LIN {X 0,Y 519.918,Z 580.66,A -85,B 0,C 180,E1 4894.132,E2 4894.132} C_VEL
LIN {X 0,Y 514.444,Z 580.66,A -85,B 0,C 180,E1 4896.247,E2 4896.247} C_VEL
LIN {X 0,Y 514.337,Z 580.66,A -85,B 0,C 180,E1 4896.492,E2 4896.492} C_VEL
LIN {X 0,Y 514.405,Z 580.66,A -85,B 0,C 180,E1 4902.622,E2 4902.622} C_VEL
LIN {X 0,Y 514.476,Z 580.66,A -85,B 0,C 180,E1 4907.4,E2 4907.4} C_VEL
LIN {X 0,Y 514.455,Z 580.66,A -85,B 0,C 180,E1 4912.61,E2 4912.61} C_VEL
LIN {X 0,Y 514.587,Z 580.66,A -85,B 0,C 180,E1 4919.328,E2 4919.328} C_VEL
LIN {X 0,Y 526.153,Z 611.087,A -85,B 0,C 180,E1 4920.404,E2 4920.404} C_VEL
LIN {X 0,Y 525.371,Z 668.245,A -85,B 0,C 180,E1 4921.362,E2 4921.362} C_VEL
LIN {X 0,Y 524.09,Z 703.782,A -85,B 0,C 180,E1 4922.574,E2 4922.574} C_VEL
LIN {X 0,Y 522.217,Z 738.252,A -85,B 0,C 180,E1 4924.451,E2 4924.451} C_VEL
LIN {X 0,Y 520.217,Z 769.927,A -85,B 0,C 180,E1 4926.884,E2 4926.884} C_VEL
LIN {X 0,Y 518.339,Z 798.982,A -85,B 0,C 180,E1 4929.926,E2 4929.926} C_VEL
LIN {X 0,Y 516.846,Z 823.631,A -85,B 0,C 180,E1 4933.403,E2 4933.403} C_VEL
LIN {X 0,Y 515.936,Z 843.713,A -85,B 0,C 180,E1 4937.284,E2 4937.284} C_VEL
LIN {X 0,Y 515.52,Z 857.455,A -85,B 0,C 180,E1 4941.129,E2 4941.129} C_VEL
LIN {X 0,Y 515.31,Z 865.962,A -85,B 0,C 180,E1 4944.942,E2 4944.942} C_VEL
LIN {X 0,Y 515.232,Z 869.509,A -85,B 0,C 180,E1 4948.315,E2 4948.315} C_VEL
LIN {X 0,Y 515.241,Z 868.974,A -85,B 0,C 180,E1 4952.558,E2 4952.558} C_VEL
LIN {X 0,Y 515.34,Z 862.769,A -85,B 0,C 180,E1 4956.747,E2 4956.747} C_VEL
LIN {X 0,Y 515.644,Z 851.662,A -85,B 0,C 180,E1 4960.67,E2 4960.67} C_VEL
LIN {X 0,Y 516.365,Z 834.554,A -85,B 0,C 180,E1 4964.646,E2 4964.646} C_VEL
LIN {X 0,Y 517.565,Z 811.69,A -85,B 0,C 180,E1 4968.416,E2 4968.416} C_VEL
LIN {X 0,Y 519.291,Z 784.441,A -85,B 0,C 180,E1 4971.705,E2 4971.705} C_VEL
LIN {X 0,Y 521.3,Z 753.854,A -85,B 0,C 180,E1 4974.446,E2 4974.446} C_VEL
LIN {X 0,Y 523.322,Z 718.255,A -85,B 0,C 180,E1 4976.729,E2 4976.729} C_VEL
LIN {X 0,Y 524.952,Z 684.31,A -85,B 0,C 180,E1 4978.166,E2 4978.166} C_VEL
LIN {X 0,Y 525.974,Z 647.659,A -85,B 0,C 180,E1 4979.056,E2 4979.056} C_VEL
LIN {X 0,Y 525.542,Z 607.493,A -85,B 0,C 180,E1 4979.68,E2 4979.68} C_VEL
LIN {X 0,Y 514.561,Z 580.66,A -85,B 0,C 180,E1 4980.717,E2 4980.717} C_VEL
LIN {X 0,Y 514.384,Z 580.66,A -85,B 0,C 180,E1 4986.061,E2 4986.061} C_VEL
LIN {X 0,Y 514.383,Z 580.66,A -85,B 0,C 180,E1 4992.628,E2 4992.628} C_VEL
LIN {X 0,Y 514.482,Z 580.66,A -85,B 0,C 180,E1 4997.409,E2 4997.409} C_VEL
LIN {X 0,Y 514.444,Z 580.66,A -85,B 0,C 180,E1 5002.616,E2 5002.616} C_VEL
LIN {X 0,Y 514.468,Z 580.66,A -85,B 0,C 180,E1 5008.584,E2 5008.584} C_VEL
LIN {X 0,Y 514.582,Z 580.66,A -85,B 0,C 180,E1 5013.816,E2 5013.816} C_VEL
LIN {X 0,Y 514.736,Z 580.66,A -85,B 0,C 180,E1 5020.255,E2 5020.255} C_VEL
LIN {X 0,Y 514.546,Z 580.66,A -85,B 0,C 180,E1 5026.162,E2 5026.162} C_VEL
LIN {X 0,Y 514.797,Z 580.66,A -85,B 0,C 180,E1 5031.549,E2 5031.549} C_VEL
LIN {X 0,Y 514.928,Z 580.66,A -85,B 0,C 180,E1 5036.633,E2 5036.633} C_VEL
LIN {X 0,Y 514.976,Z 580.66,A -85,B 0,C 180,E1 5041.689,E2 5041.689} C_VEL
LIN {X 0,Y 514.853,Z 580.66,A -85,B 0,C 180,E1 5046.76,E2 5046.76} C_VEL
LIN {X 0,Y 514.756,Z 580.66,A -85,B 0,C 180,E1 5051.886,E2 5051.886} C_VEL
LIN {X 0,Y 514.721,Z 580.66,A -85,B 0,C 180,E1 5057.111,E2 5057.111} C_VEL
LIN {X 0,Y 514.634,Z 580.66,A -85,B 0,C 180,E1 5062.491,E2 5062.491} C_VEL
LIN {X 0,Y 514.5,Z 580.66,A -85,B 0,C 180,E1 5068.094,E2 5068.094} C_VEL
LIN {X 0,Y 514.512,Z 580.66,A -85,B 0,C 180,E1 5073.999,E2 5073.999} C_VEL
LIN {X 0,Y 514.466,Z 580.66,A -85,B 0,C 180,E1 5080.082,E2 5080.082} C_VEL
LIN {X 0,Y 514.257,Z 580.66,A -85,B 0,C 180,E1 5085.045,E2 5085.045} C_VEL
LIN {X 0,Y 514.476,Z 580.66,A -85,B 0,C 180,E1 5089.927,E2 5089.927} C_VEL
LIN {X 0,Y 514.559,Z 580.66,A -85,B 0,C 180,E1 5096.012,E2 5096.012} C_VEL
LIN {X 0,Y 514.48,Z 580.66,A -85,B 0,C 180,E1 5101.998,E2 5101.998} C_VEL
LIN {X 0,Y 514.717,Z 581.391,A -85,B 0,C 180,E1 5106.325,E2 5106.325} C_VEL
LIN {X 0,Y 522.294,Z 605.692,A -85,B 0,C 180,E1 5108.079,E2 5108.079} C_VEL
LIN {X 0,Y 520.619,Z 636.027,A -85,B 0,C 180,E1 5110.242,E2 5110.242} C_VEL
LIN {X 0,Y 518.756,Z 661.49,A -85,B 0,C 180,E1 5112.836,E2 5112.836} C_VEL
LIN {X 0,Y 517.145,Z 684.027,A -85,B 0,C 180,E1 5116.042,E2 5116.042} C_VEL
LIN {X 0,Y 516.14,Z 701.171,A -85,B 0,C 180,E1 5119.522,E2 5119.522} C_VEL
LIN {X 0,Y 515.634,Z 713.151,A -85,B 0,C 180,E1 5123.257,E2 5123.257} C_VEL
LIN {X 0,Y 515.417,Z 719.891,A -85,B 0,C 180,E1 5127.222,E2 5127.222} C_VEL
LIN {X 0,Y 515.407,Z 721.257,A -85,B 0,C 180,E1 5130.002,E2 5130.002} C_VEL
LIN {X 0,Y 515.483,Z 718.032,A -85,B 0,C 180,E1 5134.212,E2 5134.212} C_VEL
LIN {X 0,Y 515.769,Z 709.434,A -85,B 0,C 180,E1 5138.017,E2 5138.017} C_VEL
LIN {X 0,Y 516.485,Z 694.755,A -85,B 0,C 180,E1 5141.843,E2 5141.843} C_VEL
LIN {X 0,Y 517.776,Z 675.211,A -85,B 0,C 180,E1 5145.26,E2 5145.26} C_VEL
LIN {X 0,Y 519.442,Z 651.913,A -85,B 0,C 180,E1 5148.152,E2 5148.152} C_VEL
LIN {X 0,Y 521.339,Z 625.142,A -85,B 0,C 180,E1 5150.533,E2 5150.533} C_VEL
LIN {X 0,Y 521.725,Z 602.202,A -85,B 0,C 180,E1 5152.079,E2 5152.079} C_VEL
LIN {X 0,Y 514.687,Z 580.66,A -85,B 0,C 180,E1 5153.646,E2 5153.646} C_VEL
LIN {X 0,Y 514.448,Z 580.66,A -85,B 0,C 180,E1 5160.022,E2 5160.022} C_VEL
LIN {X 0,Y 514.456,Z 580.66,A -85,B 0,C 180,E1 5166.059,E2 5166.059} C_VEL
LIN {X 0,Y 514.454,Z 580.66,A -85,B 0,C 180,E1 5170.352,E2 5170.352} C_VEL
LIN {X 0,Y 514.383,Z 580.66,A -85,B 0,C 180,E1 5175.05,E2 5175.05} C_VEL
LIN {X 0,Y 514.436,Z 580.66,A -85,B 0,C 180,E1 5179.927,E2 5179.927} C_VEL
LIN {X 0,Y 514.363,Z 580.66,A -85,B 0,C 180,E1 5185.989,E2 5185.989} C_VEL
LIN {X 0,Y 514.485,Z 580.66,A -85,B 0,C 180,E1 5191.99,E2 5191.99} C_VEL
LIN {X 0,Y 514.66,Z 580.66,A -85,B 0,C 180,E1 5197.51,E2 5197.51} C_VEL
LIN {X 0,Y 514.744,Z 580.66,A -85,B 0,C 180,E1 5202.89,E2 5202.89} C_VEL
LIN {X 0,Y 514.749,Z 580.66,A -85,B 0,C 180,E1 5209.831,E2 5209.831} C_VEL
LIN {X 0,Y 514.979,Z 580.66,A -85,B 0,C 180,E1 5214.935,E2 5214.935} C_VEL
LIN {X 0,Y 515.032,Z 580.66,A -85,B 0,C 180,E1 5219.995,E2 5219.995} C_VEL
LIN {X 0,Y 514.945,Z 580.66,A -85,B 0,C 180,E1 5225.056,E2 5225.056} C_VEL
LIN {X 0,Y 514.862,Z 580.66,A -85,B 0,C 180,E1 5230.158,E2 5230.158} C_VEL
LIN {X 0,Y 514.764,Z 580.66,A -85,B 0,C 180,E1 5235.345,E2 5235.345} C_VEL
LIN {X 0,Y 514.669,Z 580.66,A -85,B 0,C 180,E1 5240.666,E2 5240.666} C_VEL
LIN {X 0,Y 514.547,Z 580.66,A -85,B 0,C 180,E1 5246.186,E2 5246.186} C_VEL
LIN {X 0,Y 514.468,Z 580.66,A -85,B 0,C 180,E1 5251.981,E2 5251.981} C_VEL
LIN {X 0,Y 514.337,Z 580.66,A -85,B 0,C 180,E1 5256.492,E2 5256.492} C_VEL
LIN {X 0,Y 513.032,Z 580.66,A -85,B 0,C 180,E1 5257.458,E2 5257.458} C_VEL
LIN {X 0,Y 506.4,Z 580.66,A -85,B 0,C 180,E1 5260.09,E2 5260.09} C_VEL
LIN {X 0,Y 506.318,Z 580.66,A -85,B 0,C 180,E1 5260.34,E2 5260.34} C_VEL
LIN {X 0,Y 506.489,Z 580.66,A -85,B 0,C 180,E1 5266.563,E2 5266.563} C_VEL
LIN {X 0,Y 506.522,Z 580.66,A -85,B 0,C 180,E1 5273.285,E2 5273.285} C_VEL
LIN {X 0,Y 506.623,Z 580.66,A -85,B 0,C 180,E1 5278.911,E2 5278.911} C_VEL
LIN {X 0,Y 518.95,Z 611.439,A -85,B 0,C 180,E1 5280.047,E2 5280.047} C_VEL
LIN {X 0,Y 518.154,Z 666.942,A -85,B 0,C 180,E1 5280.995,E2 5280.995} C_VEL
LIN {X 0,Y 516.676,Z 704.173,A -85,B 0,C 180,E1 5282.276,E2 5282.276} C_VEL
LIN {X 0,Y 514.856,Z 739.728,A -85,B 0,C 180,E1 5284.176,E2 5284.176} C_VEL
LIN {X 0,Y 512.715,Z 771.394,A -85,B 0,C 180,E1 5286.662,E2 5286.662} C_VEL
LIN {X 0,Y 510.658,Z 800.734,A -85,B 0,C 180,E1 5289.837,E2 5289.837} C_VEL
LIN {X 0,Y 509.045,Z 824.956,A -85,B 0,C 180,E1 5293.364,E2 5293.364} C_VEL
LIN {X 0,Y 508.133,Z 843.713,A -85,B 0,C 180,E1 5297.086,E2 5297.086} C_VEL
LIN {X 0,Y 507.653,Z 857.481,A -85,B 0,C 180,E1 5301,E2 5301} C_VEL
LIN {X 0,Y 507.414,Z 865.961,A -85,B 0,C 180,E1 5304.863,E2 5304.863} C_VEL
LIN {X 0,Y 507.351,Z 869.51,A -85,B 0,C 180,E1 5308.288,E2 5308.288} C_VEL
LIN {X 0,Y 507.414,Z 869.512,A -85,B 0,C 180,E1 5311.708,E2 5311.708} C_VEL
LIN {X 0,Y 507.418,Z 864.456,A -85,B 0,C 180,E1 5315.993,E2 5315.993} C_VEL
LIN {X 0,Y 507.659,Z 854.965,A -85,B 0,C 180,E1 5319.832,E2 5319.832} C_VEL
LIN {X 0,Y 508.272,Z 839.833,A -85,B 0,C 180,E1 5323.785,E2 5323.785} C_VEL
LIN {X 0,Y 509.412,Z 818.483,A -85,B 0,C 180,E1 5327.691,E2 5327.691} C_VEL
LIN {X 0,Y 511.093,Z 793.355,A -85,B 0,C 180,E1 5331.057,E2 5331.057} C_VEL
LIN {X 0,Y 513.309,Z 763.038,A -85,B 0,C 180,E1 5334.075,E2 5334.075} C_VEL
LIN {X 0,Y 515.376,Z 731.713,A -85,B 0,C 180,E1 5336.323,E2 5336.323} C_VEL
LIN {X 0,Y 517.147,Z 695.545,A -85,B 0,C 180,E1 5338.079,E2 5338.079} C_VEL
LIN {X 0,Y 518.453,Z 658.867,A -85,B 0,C 180,E1 5339.19,E2 5339.19} C_VEL
LIN {X 0,Y 518.382,Z 609.73,A -85,B 0,C 180,E1 5340.008,E2 5340.008} C_VEL
LIN {X 0,Y 506.626,Z 580.66,A -85,B 0,C 180,E1 5341.084,E2 5341.084} C_VEL
LIN {X 0,Y 506.455,Z 580.66,A -85,B 0,C 180,E1 5346.717,E2 5346.717} C_VEL
LIN {X 0,Y 506.434,Z 580.66,A -85,B 0,C 180,E1 5353.438,E2 5353.438} C_VEL
LIN {X 0,Y 506.488,Z 580.66,A -85,B 0,C 180,E1 5358.886,E2 5358.886} C_VEL
LIN {X 0,Y 506.475,Z 580.66,A -85,B 0,C 180,E1 5365.397,E2 5365.397} C_VEL
LIN {X 0,Y 506.544,Z 580.66,A -85,B 0,C 180,E1 5371.436,E2 5371.436} C_VEL
LIN {X 0,Y 506.713,Z 580.66,A -85,B 0,C 180,E1 5377.854,E2 5377.854} C_VEL
LIN {X 0,Y 506.883,Z 580.66,A -85,B 0,C 180,E1 5382.899,E2 5382.899} C_VEL
LIN {X 0,Y 506.859,Z 580.66,A -85,B 0,C 180,E1 5389.68,E2 5389.68} C_VEL
LIN {X 0,Y 507.037,Z 580.66,A -85,B 0,C 180,E1 5394.865,E2 5394.865} C_VEL
LIN {X 0,Y 507.151,Z 580.66,A -85,B 0,C 180,E1 5400.005,E2 5400.005} C_VEL
LIN {X 0,Y 507.026,Z 580.66,A -85,B 0,C 180,E1 5405.144,E2 5405.144} C_VEL
LIN {X 0,Y 506.922,Z 580.66,A -85,B 0,C 180,E1 5410.328,E2 5410.328} C_VEL
LIN {X 0,Y 506.825,Z 580.66,A -85,B 0,C 180,E1 5415.601,E2 5415.601} C_VEL
LIN {X 0,Y 506.725,Z 580.66,A -85,B 0,C 180,E1 5421.016,E2 5421.016} C_VEL
LIN {X 0,Y 506.598,Z 580.66,A -85,B 0,C 180,E1 5426.639,E2 5426.639} C_VEL
LIN {X 0,Y 506.565,Z 580.66,A -85,B 0,C 180,E1 5432.552,E2 5432.552} C_VEL
LIN {X 0,Y 506.585,Z 580.66,A -85,B 0,C 180,E1 5436.714,E2 5436.714} C_VEL
LIN {X 0,Y 506.392,Z 580.66,A -85,B 0,C 180,E1 5441.632,E2 5441.632} C_VEL
LIN {X 0,Y 506.398,Z 580.66,A -85,B 0,C 180,E1 5448.377,E2 5448.377} C_VEL
LIN {X 0,Y 506.644,Z 580.66,A -85,B 0,C 180,E1 5453.798,E2 5453.798} C_VEL
LIN {X 0,Y 506.605,Z 580.66,A -85,B 0,C 180,E1 5460.085,E2 5460.085} C_VEL
LIN {X 0,Y 506.739,Z 581.087,A -85,B 0,C 180,E1 5465.795,E2 5465.795} C_VEL
LIN {X 0,Y 515.338,Z 608.137,A -85,B 0,C 180,E1 5467.767,E2 5467.767} C_VEL
LIN {X 0,Y 513.45,Z 638.063,A -85,B 0,C 180,E1 5469.955,E2 5469.955} C_VEL
LIN {X 0,Y 511.415,Z 663.071,A -85,B 0,C 180,E1 5472.559,E2 5472.559} C_VEL
LIN {X 0,Y 509.742,Z 684.128,A -85,B 0,C 180,E1 5475.585,E2 5475.585} C_VEL
LIN {X 0,Y 508.574,Z 700.614,A -85,B 0,C 180,E1 5478.898,E2 5478.898} C_VEL
LIN {X 0,Y 507.916,Z 713.339,A -85,B 0,C 180,E1 5482.723,E2 5482.723} C_VEL
LIN {X 0,Y 507.689,Z 720.49,A -85,B 0,C 180,E1 5486.582,E2 5486.582} C_VEL
LIN {X 0,Y 507.605,Z 722.443,A -85,B 0,C 180,E1 5490.002,E2 5490.002} C_VEL
LIN {X 0,Y 507.69,Z 719.247,A -85,B 0,C 180,E1 5494.277,E2 5494.277} C_VEL
LIN {X 0,Y 508.033,Z 710.734,A -85,B 0,C 180,E1 5498.14,E2 5498.14} C_VEL
LIN {X 0,Y 508.862,Z 696.187,A -85,B 0,C 180,E1 5502.023,E2 5502.023} C_VEL
LIN {X 0,Y 510.322,Z 676.833,A -85,B 0,C 180,E1 5505.488,E2 5505.488} C_VEL
LIN {X 0,Y 512.3,Z 652.382,A -85,B 0,C 180,E1 5508.573,E2 5508.573} C_VEL
LIN {X 0,Y 514.331,Z 625.587,A -85,B 0,C 180,E1 5510.965,E2 5510.965} C_VEL
LIN {X 0,Y 514.91,Z 605.372,A -85,B 0,C 180,E1 5512.348,E2 5512.348} C_VEL
LIN {X 0,Y 506.754,Z 580.66,A -85,B 0,C 180,E1 5514.15,E2 5514.15} C_VEL
LIN {X 0,Y 506.533,Z 580.66,A -85,B 0,C 180,E1 5520.541,E2 5520.541} C_VEL
LIN {X 0,Y 506.559,Z 580.66,A -85,B 0,C 180,E1 5526.712,E2 5526.712} C_VEL
LIN {X 0,Y 506.415,Z 580.66,A -85,B 0,C 180,E1 5533.445,E2 5533.445} C_VEL
LIN {X 0,Y 506.445,Z 580.66,A -85,B 0,C 180,E1 5538.869,E2 5538.869} C_VEL
LIN {X 0,Y 506.451,Z 580.66,A -85,B 0,C 180,E1 5545.383,E2 5545.383} C_VEL
LIN {X 0,Y 506.509,Z 580.66,A -85,B 0,C 180,E1 5551.423,E2 5551.423} C_VEL
LIN {X 0,Y 506.755,Z 580.66,A -85,B 0,C 180,E1 5557.851,E2 5557.851} C_VEL
LIN {X 0,Y 506.834,Z 580.66,A -85,B 0,C 180,E1 5562.927,E2 5562.927} C_VEL
LIN {X 0,Y 506.849,Z 580.66,A -85,B 0,C 180,E1 5569.67,E2 5569.67} C_VEL
LIN {X 0,Y 507.071,Z 580.66,A -85,B 0,C 180,E1 5574.856,E2 5574.856} C_VEL
LIN {X 0,Y 507.152,Z 580.66,A -85,B 0,C 180,E1 5579.995,E2 5579.995} C_VEL
LIN {X 0,Y 507.031,Z 580.66,A -85,B 0,C 180,E1 5585.135,E2 5585.135} C_VEL
LIN {X 0,Y 506.935,Z 580.66,A -85,B 0,C 180,E1 5590.318,E2 5590.318} C_VEL
LIN {X 0,Y 506.83,Z 580.66,A -85,B 0,C 180,E1 5595.591,E2 5595.591} C_VEL
LIN {X 0,Y 506.724,Z 580.66,A -85,B 0,C 180,E1 5601.006,E2 5601.006} C_VEL
LIN {X 0,Y 506.603,Z 580.66,A -85,B 0,C 180,E1 5606.629,E2 5606.629} C_VEL
LIN {X 0,Y 506.484,Z 580.66,A -85,B 0,C 180,E1 5612.547,E2 5612.547} C_VEL
LIN {X 0,Y 506.454,Z 580.66,A -85,B 0,C 180,E1 5616.713,E2 5616.713} C_VEL
LIN {X 0,Y 506.318,Z 580.66,A -85,B 0,C 180,E1 5620.34,E2 5620.34} C_VEL
LIN {X 0,Y 503.848,Z 580.66,A -85,B 0,C 180,E1 5621.801,E2 5621.801} C_VEL
LIN {X 0,Y 498.614,Z 580.66,A -85,B 0,C 180,E1 5623.992,E2 5623.992} C_VEL
LIN {X 0,Y 498.541,Z 580.66,A -85,B 0,C 180,E1 5624.245,E2 5624.245} C_VEL
LIN {X 0,Y 498.526,Z 580.66,A -85,B 0,C 180,E1 5630.372,E2 5630.372} C_VEL
LIN {X 0,Y 498.577,Z 580.66,A -85,B 0,C 180,E1 5636.864,E2 5636.864} C_VEL
LIN {X 0,Y 498.734,Z 581.255,A -85,B 0,C 180,E1 5638.488,E2 5638.488} C_VEL
LIN {X 0,Y 511.793,Z 613.809,A -85,B 0,C 180,E1 5639.711,E2 5639.711} C_VEL
LIN {X 0,Y 510.896,Z 666.664,A -85,B 0,C 180,E1 5640.644,E2 5640.644} C_VEL
LIN {X 0,Y 509.253,Z 703.957,A -85,B 0,C 180,E1 5641.957,E2 5641.957} C_VEL
LIN {X 0,Y 507.211,Z 741.098,A -85,B 0,C 180,E1 5643.995,E2 5643.995} C_VEL
LIN {X 0,Y 505.142,Z 773.341,A -85,B 0,C 180,E1 5646.509,E2 5646.509} C_VEL
LIN {X 0,Y 503.055,Z 800.734,A -85,B 0,C 180,E1 5649.519,E2 5649.519} C_VEL
LIN {X 0,Y 501.323,Z 824.954,A -85,B 0,C 180,E1 5653.1,E2 5653.1} C_VEL
LIN {X 0,Y 500.313,Z 843.712,A -85,B 0,C 180,E1 5656.88,E2 5656.88} C_VEL
LIN {X 0,Y 499.77,Z 857.604,A -85,B 0,C 180,E1 5660.904,E2 5660.904} C_VEL
LIN {X 0,Y 499.526,Z 865.961,A -85,B 0,C 180,E1 5664.781,E2 5664.781} C_VEL
LIN {X 0,Y 499.464,Z 869.509,A -85,B 0,C 180,E1 5668.261,E2 5668.261} C_VEL
LIN {X 0,Y 499.537,Z 869.511,A -85,B 0,C 180,E1 5671.735,E2 5671.735} C_VEL
LIN {X 0,Y 499.549,Z 864.455,A -85,B 0,C 180,E1 5676.088,E2 5676.088} C_VEL
LIN {X 0,Y 499.798,Z 855.024,A -85,B 0,C 180,E1 5679.969,E2 5679.969} C_VEL
LIN {X 0,Y 500.484,Z 839.833,A -85,B 0,C 180,E1 5684.003,E2 5684.003} C_VEL
LIN {X 0,Y 501.752,Z 818.482,A -85,B 0,C 180,E1 5687.97,E2 5687.97} C_VEL
LIN {X 0,Y 503.728,Z 792.238,A -85,B 0,C 180,E1 5691.514,E2 5691.514} C_VEL
LIN {X 0,Y 505.587,Z 766.202,A -85,B 0,C 180,E1 5694.118,E2 5694.118} C_VEL
LIN {X 0,Y 507.818,Z 732.007,A -85,B 0,C 180,E1 5696.575,E2 5696.575} C_VEL
LIN {X 0,Y 509.739,Z 696.218,A -85,B 0,C 180,E1 5698.372,E2 5698.372} C_VEL
LIN {X 0,Y 511.195,Z 659.434,A -85,B 0,C 180,E1 5699.528,E2 5699.528} C_VEL
LIN {X 0,Y 511.106,Z 611.816,A -85,B 0,C 180,E1 5700.355,E2 5700.355} C_VEL
LIN {X 0,Y 498.704,Z 580.66,A -85,B 0,C 180,E1 5701.606,E2 5701.606} C_VEL
LIN {X 0,Y 498.444,Z 580.66,A -85,B 0,C 180,E1 5707.846,E2 5707.846} C_VEL
LIN {X 0,Y 498.546,Z 580.66,A -85,B 0,C 180,E1 5714.303,E2 5714.303} C_VEL
LIN {X 0,Y 498.521,Z 580.66,A -85,B 0,C 180,E1 5720.38,E2 5720.38} C_VEL
LIN {X 0,Y 498.566,Z 580.66,A -85,B 0,C 180,E1 5726.871,E2 5726.871} C_VEL
LIN {X 0,Y 498.653,Z 580.66,A -85,B 0,C 180,E1 5732.912,E2 5732.912} C_VEL
LIN {X 0,Y 498.831,Z 580.66,A -85,B 0,C 180,E1 5738.646,E2 5738.646} C_VEL
LIN {X 0,Y 498.825,Z 580.66,A -85,B 0,C 180,E1 5744.152,E2 5744.152} C_VEL
LIN {X 0,Y 498.927,Z 580.66,A -85,B 0,C 180,E1 5749.514,E2 5749.514} C_VEL
LIN {X 0,Y 499.147,Z 580.66,A -85,B 0,C 180,E1 5754.784,E2 5754.784} C_VEL
LIN {X 0,Y 499.264,Z 580.66,A -85,B 0,C 180,E1 5760.005,E2 5760.005} C_VEL
LIN {X 0,Y 499.132,Z 580.66,A -85,B 0,C 180,E1 5765.226,E2 5765.226} C_VEL
LIN {X 0,Y 498.993,Z 580.66,A -85,B 0,C 180,E1 5770.494,E2 5770.494} C_VEL
LIN {X 0,Y 498.908,Z 580.66,A -85,B 0,C 180,E1 5775.855,E2 5775.855} C_VEL
LIN {X 0,Y 498.819,Z 580.66,A -85,B 0,C 180,E1 5781.365,E2 5781.365} C_VEL
LIN {X 0,Y 498.633,Z 580.66,A -85,B 0,C 180,E1 5787.1,E2 5787.1} C_VEL
LIN {X 0,Y 498.673,Z 580.66,A -85,B 0,C 180,E1 5793.133,E2 5793.133} C_VEL
LIN {X 0,Y 498.513,Z 580.66,A -85,B 0,C 180,E1 5799.633,E2 5799.633} C_VEL
LIN {X 0,Y 498.387,Z 580.66,A -85,B 0,C 180,E1 5805.679,E2 5805.679} C_VEL
LIN {X 0,Y 498.583,Z 580.66,A -85,B 0,C 180,E1 5812.15,E2 5812.15} C_VEL
LIN {X 0,Y 498.669,Z 580.66,A -85,B 0,C 180,E1 5818.234,E2 5818.234} C_VEL
LIN {X 0,Y 498.714,Z 580.66,A -85,B 0,C 180,E1 5825.056,E2 5825.056} C_VEL
LIN {X 0,Y 498.731,Z 580.937,A -85,B 0,C 180,E1 5825.262,E2 5825.262} C_VEL
LIN {X 0,Y 508.286,Z 610.371,A -85,B 0,C 180,E1 5827.44,E2 5827.44} C_VEL
LIN {X 0,Y 506.283,Z 640.066,A -85,B 0,C 180,E1 5829.659,E2 5829.659} C_VEL
LIN {X 0,Y 504.07,Z 665.141,A -85,B 0,C 180,E1 5832.333,E2 5832.333} C_VEL
LIN {X 0,Y 502.086,Z 687.362,A -85,B 0,C 180,E1 5835.665,E2 5835.665} C_VEL
LIN {X 0,Y 500.816,Z 703.745,A -85,B 0,C 180,E1 5839.154,E2 5839.154} C_VEL
LIN {X 0,Y 500.13,Z 715.672,A -85,B 0,C 180,E1 5843.047,E2 5843.047} C_VEL
LIN {X 0,Y 499.899,Z 721.697,A -85,B 0,C 180,E1 5846.529,E2 5846.529} C_VEL
LIN {X 0,Y 499.816,Z 723.626,A -85,B 0,C 180,E1 5850.002,E2 5850.002} C_VEL
LIN {X 0,Y 499.93,Z 720.461,A -85,B 0,C 180,E1 5854.344,E2 5854.344} C_VEL
LIN {X 0,Y 500.309,Z 712.03,A -85,B 0,C 180,E1 5858.266,E2 5858.266} C_VEL
LIN {X 0,Y 501.267,Z 697.633,A -85,B 0,C 180,E1 5862.208,E2 5862.208} C_VEL
LIN {X 0,Y 502.908,Z 678.494,A -85,B 0,C 180,E1 5865.722,E2 5865.722} C_VEL
LIN {X 0,Y 505.019,Z 654.517,A -85,B 0,C 180,E1 5868.821,E2 5868.821} C_VEL
LIN {X 0,Y 507.222,Z 627.716,A -85,B 0,C 180,E1 5871.276,E2 5871.276} C_VEL
LIN {X 0,Y 507.625,Z 607.027,A -85,B 0,C 180,E1 5872.728,E2 5872.728} C_VEL
LIN {X 0,Y 498.785,Z 580.66,A -85,B 0,C 180,E1 5874.739,E2 5874.739} C_VEL
LIN {X 0,Y 498.552,Z 580.66,A -85,B 0,C 180,E1 5881.084,E2 5881.084} C_VEL
LIN {X 0,Y 498.563,Z 580.66,A -85,B 0,C 180,E1 5887.4,E2 5887.4} C_VEL
LIN {X 0,Y 498.52,Z 580.66,A -85,B 0,C 180,E1 5893.199,E2 5893.199} C_VEL
LIN {X 0,Y 498.477,Z 580.66,A -85,B 0,C 180,E1 5899.407,E2 5899.407} C_VEL
LIN {X 0,Y 498.545,Z 580.66,A -85,B 0,C 180,E1 5905.083,E2 5905.083} C_VEL
LIN {X 0,Y 498.589,Z 580.66,A -85,B 0,C 180,E1 5911.72,E2 5911.72} C_VEL
LIN {X 0,Y 498.777,Z 580.66,A -85,B 0,C 180,E1 5916.753,E2 5916.753} C_VEL
LIN {X 0,Y 498.9,Z 580.66,A -85,B 0,C 180,E1 5922.329,E2 5922.329} C_VEL
LIN {X 0,Y 498.777,Z 580.66,A -85,B 0,C 180,E1 5927.727,E2 5927.727} C_VEL
LIN {X 0,Y 499.161,Z 580.66,A -85,B 0,C 180,E1 5933.026,E2 5933.026} C_VEL
LIN {X 0,Y 499.406,Z 580.66,A -85,B 0,C 180,E1 5938.258,E2 5938.258} C_VEL
LIN {X 0,Y 499.278,Z 580.66,A -85,B 0,C 180,E1 5943.472,E2 5943.472} C_VEL
LIN {X 0,Y 499.087,Z 580.66,A -85,B 0,C 180,E1 5948.719,E2 5948.719} C_VEL
LIN {X 0,Y 498.964,Z 580.66,A -85,B 0,C 180,E1 5954.044,E2 5954.044} C_VEL
LIN {X 0,Y 498.82,Z 580.66,A -85,B 0,C 180,E1 5959.79,E2 5959.79} C_VEL
LIN {X 0,Y 498.729,Z 580.66,A -85,B 0,C 180,E1 5965.146,E2 5965.146} C_VEL
LIN {X 0,Y 498.556,Z 580.66,A -85,B 0,C 180,E1 5971.752,E2 5971.752} C_VEL
LIN {X 0,Y 498.449,Z 580.66,A -85,B 0,C 180,E1 5977.836,E2 5977.836} C_VEL
LIN {X 0,Y 498.541,Z 580.66,A -85,B 0,C 180,E1 5984.245,E2 5984.245} C_VEL
LIN {X 0,Y 496.111,Z 580.66,A -85,B 0,C 180,E1 5985.721,E2 5985.721} C_VEL
LIN {X 0,Y 490.617,Z 580.66,A -85,B 0,C 180,E1 5988.19,E2 5988.19} C_VEL
LIN {X 0,Y 490.592,Z 580.66,A -85,B 0,C 180,E1 5994.099,E2 5994.099} C_VEL
LIN {X 0,Y 490.78,Z 581.184,A -85,B 0,C 180,E1 5998.017,E2 5998.017} C_VEL
LIN {X 0,Y 504.572,Z 615.556,A -85,B 0,C 180,E1 5999.357,E2 5999.357} C_VEL
LIN {X 0,Y 503.668,Z 666.13,A -85,B 0,C 180,E1 6000.277,E2 6000.277} C_VEL
LIN {X 0,Y 501.881,Z 703.756,A -85,B 0,C 180,E1 6001.63,E2 6001.63} C_VEL
LIN {X 0,Y 499.708,Z 740.29,A -85,B 0,C 180,E1 6003.675,E2 6003.675} C_VEL
LIN {X 0,Y 497.408,Z 773.948,A -85,B 0,C 180,E1 6006.358,E2 6006.358} C_VEL
LIN {X 0,Y 495.345,Z 802.758,A -85,B 0,C 180,E1 6009.469,E2 6009.469} C_VEL
LIN {X 0,Y 493.526,Z 826.277,A -85,B 0,C 180,E1 6013.054,E2 6013.054} C_VEL
LIN {X 0,Y 492.39,Z 845.476,A -85,B 0,C 180,E1 6017.117,E2 6017.117} C_VEL
LIN {X 0,Y 491.854,Z 858.602,A -85,B 0,C 180,E1 6021.145,E2 6021.145} C_VEL
LIN {X 0,Y 491.629,Z 867.169,A -85,B 0,C 180,E1 6025.583,E2 6025.583} C_VEL
LIN {X 0,Y 491.56,Z 870,A -85,B 0,C 180,E1 6029.998,E2 6029.998} C_VEL
LIN {X 0,Y 491.666,Z 867.175,A -85,B 0,C 180,E1 6034.414,E2 6034.414} C_VEL
LIN {X 0,Y 491.845,Z 858.607,A -85,B 0,C 180,E1 6038.852,E2 6038.852} C_VEL
LIN {X 0,Y 492.371,Z 845.488,A -85,B 0,C 180,E1 6042.88,E2 6042.88} C_VEL
LIN {X 0,Y 493.473,Z 826.295,A -85,B 0,C 180,E1 6046.944,E2 6046.944} C_VEL
LIN {X 0,Y 495.299,Z 802.814,A -85,B 0,C 180,E1 6050.525,E2 6050.525} C_VEL
LIN {X 0,Y 497.318,Z 775.112,A -85,B 0,C 180,E1 6053.533,E2 6053.533} C_VEL
LIN {X 0,Y 499.664,Z 741.808,A -85,B 0,C 180,E1 6056.216,E2 6056.216} C_VEL
LIN {X 0,Y 501.85,Z 705.126,A -85,B 0,C 180,E1 6058.306,E2 6058.306} C_VEL
LIN {X 0,Y 503.6,Z 667.94,A -85,B 0,C 180,E1 6059.672,E2 6059.672} C_VEL
LIN {X 0,Y 504.579,Z 617.97,A -85,B 0,C 180,E1 6060.61,E2 6060.61} C_VEL
LIN {X 0,Y 502.093,Z 609.835,A -85,B 0,C 180,E1 6060.875,E2 6060.875} C_VEL
LIN {X 0,Y 490.756,Z 580.66,A -85,B 0,C 180,E1 6062.037,E2 6062.037} C_VEL
LIN {X 0,Y 490.514,Z 580.66,A -85,B 0,C 180,E1 6068.119,E2 6068.119} C_VEL
LIN {X 0,Y 490.612,Z 580.66,A -85,B 0,C 180,E1 6072.757,E2 6072.757} C_VEL
LIN {X 0,Y 490.676,Z 580.66,A -85,B 0,C 180,E1 6077.775,E2 6077.775} C_VEL
LIN {X 0,Y 490.583,Z 580.66,A -85,B 0,C 180,E1 6084.106,E2 6084.106} C_VEL
LIN {X 0,Y 490.644,Z 580.66,A -85,B 0,C 180,E1 6090.42,E2 6090.42} C_VEL
LIN {X 0,Y 490.821,Z 580.66,A -85,B 0,C 180,E1 6096.364,E2 6096.364} C_VEL
LIN {X 0,Y 490.992,Z 580.66,A -85,B 0,C 180,E1 6102.045,E2 6102.045} C_VEL
LIN {X 0,Y 490.896,Z 580.66,A -85,B 0,C 180,E1 6107.537,E2 6107.537} C_VEL
LIN {X 0,Y 491.213,Z 580.66,A -85,B 0,C 180,E1 6112.923,E2 6112.923} C_VEL
LIN {X 0,Y 491.465,Z 580.66,A -85,B 0,C 180,E1 6118.24,E2 6118.24} C_VEL
LIN {X 0,Y 491.367,Z 580.66,A -85,B 0,C 180,E1 6123.538,E2 6123.538} C_VEL
LIN {X 0,Y 491.093,Z 580.66,A -85,B 0,C 180,E1 6129.419,E2 6129.419} C_VEL
LIN {X 0,Y 491.015,Z 580.66,A -85,B 0,C 180,E1 6134.286,E2 6134.286} C_VEL
LIN {X 0,Y 490.918,Z 580.66,A -85,B 0,C 180,E1 6139.836,E2 6139.836} C_VEL
LIN {X 0,Y 490.745,Z 580.66,A -85,B 0,C 180,E1 6145.595,E2 6145.595} C_VEL
LIN {X 0,Y 490.736,Z 580.66,A -85,B 0,C 180,E1 6151.639,E2 6151.639} C_VEL
LIN {X 0,Y 490.625,Z 580.66,A -85,B 0,C 180,E1 6158.117,E2 6158.117} C_VEL
LIN {X 0,Y 490.457,Z 580.66,A -85,B 0,C 180,E1 6164.767,E2 6164.767} C_VEL
LIN {X 0,Y 490.615,Z 580.66,A -85,B 0,C 180,E1 6170.496,E2 6170.496} C_VEL
LIN {X 0,Y 490.786,Z 580.66,A -85,B 0,C 180,E1 6176.409,E2 6176.409} C_VEL
LIN {X 0,Y 490.689,Z 580.66,A -85,B 0,C 180,E1 6182.432,E2 6182.432} C_VEL
LIN {X 0,Y 490.807,Z 581.125,A -85,B 0,C 180,E1 6184.738,E2 6184.738} C_VEL
LIN {X 0,Y 500.89,Z 610.698,A -85,B 0,C 180,E1 6186.976,E2 6186.976} C_VEL
LIN {X 0,Y 499.176,Z 640.64,A -85,B 0,C 180,E1 6189.24,E2 6189.24} C_VEL
LIN {X 0,Y 496.784,Z 666.617,A -85,B 0,C 180,E1 6192.031,E2 6192.031} C_VEL
LIN {X 0,Y 494.71,Z 687.755,A -85,B 0,C 180,E1 6195.231,E2 6195.231} C_VEL
LIN {X 0,Y 493.187,Z 705.132,A -85,B 0,C 180,E1 6198.985,E2 6198.985} C_VEL
LIN {X 0,Y 492.38,Z 716.947,A -85,B 0,C 180,E1 6202.937,E2 6202.937} C_VEL
LIN {X 0,Y 492.112,Z 722.904,A -85,B 0,C 180,E1 6206.474,E2 6206.474} C_VEL
LIN {X 0,Y 492.006,Z 724.813,A -85,B 0,C 180,E1 6210.002,E2 6210.002} C_VEL
LIN {X 0,Y 492.158,Z 721.676,A -85,B 0,C 180,E1 6214.412,E2 6214.412} C_VEL
LIN {X 0,Y 492.586,Z 713.346,A -85,B 0,C 180,E1 6218.397,E2 6218.397} C_VEL
LIN {X 0,Y 493.681,Z 699.095,A -85,B 0,C 180,E1 6222.398,E2 6222.398} C_VEL
LIN {X 0,Y 495.47,Z 680.148,A -85,B 0,C 180,E1 6225.965,E2 6225.965} C_VEL
LIN {X 0,Y 497.722,Z 656.599,A -85,B 0,C 180,E1 6229.069,E2 6229.069} C_VEL
LIN {X 0,Y 500.099,Z 629.58,A -85,B 0,C 180,E1 6231.594,E2 6231.594} C_VEL
LIN {X 0,Y 500.764,Z 610.335,A -85,B 0,C 180,E1 6232.964,E2 6232.964} C_VEL
LIN {X 0,Y 490.859,Z 580.66,A -85,B 0,C 180,E1 6235.296,E2 6235.296} C_VEL
LIN {X 0,Y 490.656,Z 580.66,A -85,B 0,C 180,E1 6241.641,E2 6241.641} C_VEL
LIN {X 0,Y 490.62,Z 580.66,A -85,B 0,C 180,E1 6248.113,E2 6248.113} C_VEL
LIN {X 0,Y 490.606,Z 580.66,A -85,B 0,C 180,E1 6254.775,E2 6254.775} C_VEL
LIN {X 0,Y 490.566,Z 580.66,A -85,B 0,C 180,E1 6260.497,E2 6260.497} C_VEL
LIN {X 0,Y 490.583,Z 580.66,A -85,B 0,C 180,E1 6266.438,E2 6266.438} C_VEL
LIN {X 0,Y 490.695,Z 580.66,A -85,B 0,C 180,E1 6272.425,E2 6272.425} C_VEL
LIN {X 0,Y 490.9,Z 580.66,A -85,B 0,C 180,E1 6278.273,E2 6278.273} C_VEL
LIN {X 0,Y 490.893,Z 580.66,A -85,B 0,C 180,E1 6283.879,E2 6283.879} C_VEL
LIN {X 0,Y 491.019,Z 580.66,A -85,B 0,C 180,E1 6290.653,E2 6290.653} C_VEL
LIN {X 0,Y 491.246,Z 580.66,A -85,B 0,C 180,E1 6296.461,E2 6296.461} C_VEL
LIN {X 0,Y 491.274,Z 580.66,A -85,B 0,C 180,E1 6301.761,E2 6301.761} C_VEL
LIN {X 0,Y 491.13,Z 580.66,A -85,B 0,C 180,E1 6307.078,E2 6307.078} C_VEL
LIN {X 0,Y 491.028,Z 580.66,A -85,B 0,C 180,E1 6312.46,E2 6312.46} C_VEL
LIN {X 0,Y 490.946,Z 580.66,A -85,B 0,C 180,E1 6317.957,E2 6317.957} C_VEL
LIN {X 0,Y 490.824,Z 580.66,A -85,B 0,C 180,E1 6323.636,E2 6323.636} C_VEL
LIN {X 0,Y 490.629,Z 580.66,A -85,B 0,C 180,E1 6330.223,E2 6330.223} C_VEL
LIN {X 0,Y 490.556,Z 580.66,A -85,B 0,C 180,E1 6335.896,E2 6335.896} C_VEL
LIN {X 0,Y 490.615,Z 580.66,A -85,B 0,C 180,E1 6342.212,E2 6342.212} C_VEL
LIN {X 0,Y 490.617,Z 580.66,A -85,B 0,C 180,E1 6348.19,E2 6348.19} C_VEL
LIN {X 0,Y 486.603,Z 580.66,A -85,B 0,C 180,E1 6350.173,E2 6350.173} C_VEL
LIN {X 0,Y 482.628,Z 580.66,A -85,B 0,C 180,E1 6352.188,E2 6352.188} C_VEL
LIN {X 0,Y 482.827,Z 581.081,A -85,B 0,C 180,E1 6357.525,E2 6357.525} C_VEL
LIN {X 0,Y 497.431,Z 617.812,A -85,B 0,C 180,E1 6359.009,E2 6359.009} C_VEL
LIN {X 0,Y 496.391,Z 666.424,A -85,B 0,C 180,E1 6359.931,E2 6359.931} C_VEL
LIN {X 0,Y 494.499,Z 703.413,A -85,B 0,C 180,E1 6361.293,E2 6361.293} C_VEL
LIN {X 0,Y 492.147,Z 740.201,A -85,B 0,C 180,E1 6363.397,E2 6363.397} C_VEL
LIN {X 0,Y 489.71,Z 773.499,A -85,B 0,C 180,E1 6366.107,E2 6366.107} C_VEL
LIN {X 0,Y 487.452,Z 803.883,A -85,B 0,C 180,E1 6369.464,E2 6369.464} C_VEL
LIN {X 0,Y 485.728,Z 827.46,A -85,B 0,C 180,E1 6373.007,E2 6373.007} C_VEL
LIN {X 0,Y 484.591,Z 845.476,A -85,B 0,C 180,E1 6376.906,E2 6376.906} C_VEL
LIN {X 0,Y 483.987,Z 858.602,A -85,B 0,C 180,E1 6381,E2 6381} C_VEL
LIN {X 0,Y 483.745,Z 867.168,A -85,B 0,C 180,E1 6385.511,E2 6385.511} C_VEL
LIN {X 0,Y 483.668,Z 870,A -85,B 0,C 180,E1 6389.998,E2 6389.998} C_VEL
LIN {X 0,Y 483.777,Z 867.175,A -85,B 0,C 180,E1 6394.486,E2 6394.486} C_VEL
LIN {X 0,Y 483.972,Z 858.607,A -85,B 0,C 180,E1 6398.997,E2 6398.997} C_VEL
LIN {X 0,Y 484.568,Z 845.487,A -85,B 0,C 180,E1 6403.091,E2 6403.091} C_VEL
LIN {X 0,Y 485.778,Z 826.214,A -85,B 0,C 180,E1 6407.221,E2 6407.221} C_VEL
LIN {X 0,Y 487.48,Z 802.466,A -85,B 0,C 180,E1 6410.713,E2 6410.713} C_VEL
LIN {X 0,Y 489.703,Z 773.529,A -85,B 0,C 180,E1 6413.889,E2 6413.889} C_VEL
LIN {X 0,Y 492.209,Z 740.091,A -85,B 0,C 180,E1 6416.609,E2 6416.609} C_VEL
LIN {X 0,Y 494.57,Z 703.529,A -85,B 0,C 180,E1 6418.699,E2 6418.699} C_VEL
LIN {X 0,Y 496.458,Z 665.8,A -85,B 0,C 180,E1 6420.086,E2 6420.086} C_VEL
LIN {X 0,Y 497.1,Z 616.827,A -85,B 0,C 180,E1 6421.037,E2 6421.037} C_VEL
LIN {X 0,Y 482.811,Z 580.66,A -85,B 0,C 180,E1 6422.555,E2 6422.555} C_VEL
LIN {X 0,Y 482.584,Z 580.66,A -85,B 0,C 180,E1 6428.861,E2 6428.861} C_VEL
LIN {X 0,Y 482.644,Z 580.66,A -85,B 0,C 180,E1 6433.829,E2 6433.829} C_VEL
LIN {X 0,Y 482.699,Z 580.66,A -85,B 0,C 180,E1 6438.829,E2 6438.829} C_VEL
LIN {X 0,Y 482.633,Z 580.66,A -85,B 0,C 180,E1 6444.646,E2 6444.646} C_VEL
LIN {X 0,Y 482.742,Z 580.66,A -85,B 0,C 180,E1 6449.886,E2 6449.886} C_VEL
LIN {X 0,Y 482.862,Z 580.66,A -85,B 0,C 180,E1 6455.95,E2 6455.95} C_VEL
LIN {X 0,Y 483.056,Z 580.66,A -85,B 0,C 180,E1 6461.739,E2 6461.739} C_VEL
LIN {X 0,Y 482.964,Z 580.66,A -85,B 0,C 180,E1 6467.329,E2 6467.329} C_VEL
LIN {X 0,Y 483.294,Z 580.66,A -85,B 0,C 180,E1 6472.806,E2 6472.806} C_VEL
LIN {X 0,Y 483.557,Z 580.66,A -85,B 0,C 180,E1 6478.211,E2 6478.211} C_VEL
LIN {X 0,Y 483.478,Z 580.66,A -85,B 0,C 180,E1 6483.596,E2 6483.596} C_VEL
LIN {X 0,Y 483.234,Z 580.66,A -85,B 0,C 180,E1 6489.018,E2 6489.018} C_VEL
LIN {X 0,Y 483.089,Z 580.66,A -85,B 0,C 180,E1 6494.526,E2 6494.526} C_VEL
LIN {X 0,Y 482.981,Z 580.66,A -85,B 0,C 180,E1 6500.176,E2 6500.176} C_VEL
LIN {X 0,Y 482.835,Z 580.66,A -85,B 0,C 180,E1 6506.046,E2 6506.046} C_VEL
LIN {X 0,Y 482.802,Z 580.66,A -85,B 0,C 180,E1 6512.221,E2 6512.221} C_VEL
LIN {X 0,Y 482.702,Z 580.66,A -85,B 0,C 180,E1 6518.362,E2 6518.362} C_VEL
LIN {X 0,Y 482.503,Z 580.66,A -85,B 0,C 180,E1 6523.807,E2 6523.807} C_VEL
LIN {X 0,Y 482.603,Z 580.66,A -85,B 0,C 180,E1 6528.853,E2 6528.853} C_VEL
LIN {X 0,Y 482.781,Z 580.66,A -85,B 0,C 180,E1 6534.633,E2 6534.633} C_VEL
LIN {X 0,Y 482.784,Z 580.66,A -85,B 0,C 180,E1 6539.885,E2 6539.885} C_VEL
LIN {X 0,Y 482.818,Z 580.862,A -85,B 0,C 180,E1 6544.18,E2 6544.18} C_VEL
LIN {X 0,Y 493.345,Z 611.833,A -85,B 0,C 180,E1 6546.55,E2 6546.55} C_VEL
LIN {X 0,Y 493.567,Z 623.171,A -85,B 0,C 180,E1 6547.369,E2 6547.369} C_VEL
LIN {X 0,Y 491.091,Z 651.518,A -85,B 0,C 180,E1 6549.826,E2 6549.826} C_VEL
LIN {X 0,Y 488.748,Z 674.787,A -85,B 0,C 180,E1 6552.655,E2 6552.655} C_VEL
LIN {X 0,Y 486.677,Z 694.704,A -85,B 0,C 180,E1 6556.05,E2 6556.05} C_VEL
LIN {X 0,Y 485.242,Z 710.22,A -85,B 0,C 180,E1 6559.881,E2 6559.881} C_VEL
LIN {X 0,Y 484.567,Z 720.053,A -85,B 0,C 180,E1 6563.723,E2 6563.723} C_VEL
LIN {X 0,Y 484.338,Z 724.112,A -85,B 0,C 180,E1 6566.417,E2 6566.417} C_VEL
LIN {X 0,Y 484.212,Z 725.997,A -85,B 0,C 180,E1 6570.002,E2 6570.002} C_VEL
LIN {X 0,Y 484.382,Z 722.896,A -85,B 0,C 180,E1 6574.483,E2 6574.483} C_VEL
LIN {X 0,Y 484.878,Z 714.657,A -85,B 0,C 180,E1 6578.531,E2 6578.531} C_VEL
LIN {X 0,Y 486.087,Z 700.549,A -85,B 0,C 180,E1 6582.595,E2 6582.595} C_VEL
LIN {X 0,Y 488.019,Z 681.665,A -85,B 0,C 180,E1 6586.215,E2 6586.215} C_VEL
LIN {X 0,Y 490.389,Z 658.526,A -85,B 0,C 180,E1 6589.324,E2 6589.324} C_VEL
LIN {X 0,Y 492.935,Z 631.469,A -85,B 0,C 180,E1 6591.91,E2 6591.91} C_VEL
LIN {X 0,Y 493.578,Z 612.523,A -85,B 0,C 180,E1 6593.297,E2 6593.297} C_VEL
LIN {X 0,Y 482.985,Z 581.826,A -85,B 0,C 180,E1 6595.679,E2 6595.679} C_VEL
LIN {X 0,Y 482.866,Z 580.66,A -85,B 0,C 180,E1 6595.858,E2 6595.858} C_VEL
LIN {X 0,Y 482.711,Z 580.66,A -85,B 0,C 180,E1 6602.224,E2 6602.224} C_VEL
LIN {X 0,Y 482.683,Z 580.66,A -85,B 0,C 180,E1 6608.856,E2 6608.856} C_VEL
LIN {X 0,Y 482.625,Z 580.66,A -85,B 0,C 180,E1 6613.812,E2 6613.812} C_VEL
LIN {X 0,Y 482.647,Z 580.66,A -85,B 0,C 180,E1 6618.841,E2 6618.841} C_VEL
LIN {X 0,Y 482.597,Z 580.66,A -85,B 0,C 180,E1 6624.658,E2 6624.658} C_VEL
LIN {X 0,Y 482.703,Z 580.66,A -85,B 0,C 180,E1 6629.872,E2 6629.872} C_VEL
LIN {X 0,Y 482.882,Z 580.66,A -85,B 0,C 180,E1 6635.94,E2 6635.94} C_VEL
LIN {X 0,Y 483.049,Z 580.66,A -85,B 0,C 180,E1 6641.729,E2 6641.729} C_VEL
LIN {X 0,Y 482.935,Z 580.66,A -85,B 0,C 180,E1 6647.318,E2 6647.318} C_VEL
LIN {X 0,Y 483.313,Z 580.66,A -85,B 0,C 180,E1 6652.797,E2 6652.797} C_VEL
LIN {X 0,Y 483.588,Z 580.66,A -85,B 0,C 180,E1 6658.201,E2 6658.201} C_VEL
LIN {X 0,Y 483.48,Z 580.66,A -85,B 0,C 180,E1 6663.586,E2 6663.586} C_VEL
LIN {X 0,Y 483.244,Z 580.66,A -85,B 0,C 180,E1 6669.008,E2 6669.008} C_VEL
LIN {X 0,Y 483.102,Z 580.66,A -85,B 0,C 180,E1 6674.515,E2 6674.515} C_VEL
LIN {X 0,Y 482.979,Z 580.66,A -85,B 0,C 180,E1 6680.166,E2 6680.166} C_VEL
LIN {X 0,Y 482.843,Z 580.66,A -85,B 0,C 180,E1 6686.034,E2 6686.034} C_VEL
LIN {X 0,Y 482.717,Z 580.66,A -85,B 0,C 180,E1 6692.216,E2 6692.216} C_VEL
LIN {X 0,Y 482.596,Z 580.66,A -85,B 0,C 180,E1 6698.856,E2 6698.856} C_VEL
LIN {X 0,Y 482.651,Z 580.66,A -85,B 0,C 180,E1 6703.821,E2 6703.821} C_VEL
LIN {X 0,Y 482.686,Z 580.66,A -85,B 0,C 180,E1 6708.826,E2 6708.826} C_VEL
LIN {X 0,Y 482.628,Z 580.66,A -85,B 0,C 180,E1 6712.188,E2 6712.188} C_VEL
LIN {X 0,Y 481.339,Z 580.66,A -85,B 0,C 180,E1 6713.215,E2 6713.215} C_VEL
LIN {X 0,Y 474.865,Z 580.66,A -85,B 0,C 180,E1 6716.016,E2 6716.016} C_VEL
LIN {X 0,Y 474.803,Z 580.66,A -85,B 0,C 180,E1 6716.281,E2 6716.281} C_VEL
LIN {X 0,Y 474.885,Z 580.66,A -85,B 0,C 180,E1 6716.975,E2 6716.975} C_VEL
LIN {X 0,Y 490.33,Z 621.103,A -85,B 0,C 180,E1 6718.668,E2 6718.668} C_VEL
LIN {X 0,Y 489.141,Z 666.429,A -85,B 0,C 180,E1 6719.565,E2 6719.565} C_VEL
LIN {X 0,Y 487.071,Z 703.63,A -85,B 0,C 180,E1 6720.976,E2 6720.976} C_VEL
LIN {X 0,Y 484.557,Z 740.405,A -85,B 0,C 180,E1 6723.14,E2 6723.14} C_VEL
LIN {X 0,Y 482.099,Z 772.36,A -85,B 0,C 180,E1 6725.784,E2 6725.784} C_VEL
LIN {X 0,Y 479.715,Z 802.526,A -85,B 0,C 180,E1 6729.162,E2 6729.162} C_VEL
LIN {X 0,Y 477.825,Z 827.675,A -85,B 0,C 180,E1 6732.996,E2 6732.996} C_VEL
LIN {X 0,Y 476.766,Z 845.471,A -85,B 0,C 180,E1 6736.706,E2 6736.706} C_VEL
LIN {X 0,Y 476.107,Z 858.602,A -85,B 0,C 180,E1 6740.849,E2 6740.849} C_VEL
LIN {X 0,Y 475.847,Z 867.168,A -85,B 0,C 180,E1 6745.436,E2 6745.436} C_VEL
LIN {X 0,Y 475.768,Z 870,A -85,B 0,C 180,E1 6749.998,E2 6749.998} C_VEL
LIN {X 0,Y 475.876,Z 867.174,A -85,B 0,C 180,E1 6754.56,E2 6754.56} C_VEL
LIN {X 0,Y 476.088,Z 858.606,A -85,B 0,C 180,E1 6759.148,E2 6759.148} C_VEL
LIN {X 0,Y 476.745,Z 845.458,A -85,B 0,C 180,E1 6763.297,E2 6763.297} C_VEL
LIN {X 0,Y 477.876,Z 826.461,A -85,B 0,C 180,E1 6767.222,E2 6767.222} C_VEL
LIN {X 0,Y 479.725,Z 801.244,A -85,B 0,C 180,E1 6771.001,E2 6771.001} C_VEL
LIN {X 0,Y 482.085,Z 772.297,A -85,B 0,C 180,E1 6774.223,E2 6774.223} C_VEL
LIN {X 0,Y 484.698,Z 739.198,A -85,B 0,C 180,E1 6776.945,E2 6776.945} C_VEL
LIN {X 0,Y 487.181,Z 703.356,A -85,B 0,C 180,E1 6779.033,E2 6779.033} C_VEL
LIN {X 0,Y 489.197,Z 666.097,A -85,B 0,C 180,E1 6780.443,E2 6780.443} C_VEL
LIN {X 0,Y 489.908,Z 618.957,A -85,B 0,C 180,E1 6781.401,E2 6781.401} C_VEL
LIN {X 0,Y 474.887,Z 580.66,A -85,B 0,C 180,E1 6783.089,E2 6783.089} C_VEL
LIN {X 0,Y 474.603,Z 580.66,A -85,B 0,C 180,E1 6790.046,E2 6790.046} C_VEL
LIN {X 0,Y 474.682,Z 580.66,A -85,B 0,C 180,E1 6795.443,E2 6795.443} C_VEL
LIN {X 0,Y 474.687,Z 580.66,A -85,B 0,C 180,E1 6800.371,E2 6800.371} C_VEL
LIN {X 0,Y 474.71,Z 580.66,A -85,B 0,C 180,E1 6806.017,E2 6806.017} C_VEL
LIN {X 0,Y 474.823,Z 580.66,A -85,B 0,C 180,E1 6811.432,E2 6811.432} C_VEL
LIN {X 0,Y 474.993,Z 580.66,A -85,B 0,C 180,E1 6817.568,E2 6817.568} C_VEL
LIN {X 0,Y 475.08,Z 580.66,A -85,B 0,C 180,E1 6823.338,E2 6823.338} C_VEL
LIN {X 0,Y 475.147,Z 580.66,A -85,B 0,C 180,E1 6828.983,E2 6828.983} C_VEL
LIN {X 0,Y 475.422,Z 580.66,A -85,B 0,C 180,E1 6834.523,E2 6834.523} C_VEL
LIN {X 0,Y 475.59,Z 580.66,A -85,B 0,C 180,E1 6840.005,E2 6840.005} C_VEL
LIN {X 0,Y 475.397,Z 580.66,A -85,B 0,C 180,E1 6845.488,E2 6845.488} C_VEL
LIN {X 0,Y 475.219,Z 580.66,A -85,B 0,C 180,E1 6851.026,E2 6851.026} C_VEL
LIN {X 0,Y 475.088,Z 580.66,A -85,B 0,C 180,E1 6857.057,E2 6857.057} C_VEL
LIN {X 0,Y 475.007,Z 580.66,A -85,B 0,C 180,E1 6862.493,E2 6862.493} C_VEL
LIN {X 0,Y 474.827,Z 580.66,A -85,B 0,C 180,E1 6868.579,E2 6868.579} C_VEL
LIN {X 0,Y 474.828,Z 580.66,A -85,B 0,C 180,E1 6875.032,E2 6875.032} C_VEL
LIN {X 0,Y 474.64,Z 580.66,A -85,B 0,C 180,E1 6880.046,E2 6880.046} C_VEL
LIN {X 0,Y 474.52,Z 580.66,A -85,B 0,C 180,E1 6885.42,E2 6885.42} C_VEL
LIN {X 0,Y 474.676,Z 580.66,A -85,B 0,C 180,E1 6890.366,E2 6890.366} C_VEL
LIN {X 0,Y 474.835,Z 580.66,A -85,B 0,C 180,E1 6896.007,E2 6896.007} C_VEL
LIN {X 0,Y 474.831,Z 580.66,A -85,B 0,C 180,E1 6901.429,E2 6901.429} C_VEL
LIN {X 0,Y 474.867,Z 580.66,A -85,B 0,C 180,E1 6903.605,E2 6903.605} C_VEL
LIN {X 0,Y 485.491,Z 611.768,A -85,B 0,C 180,E1 6906.012,E2 6906.012} C_VEL
LIN {X 0,Y 486.798,Z 620.329,A -85,B 0,C 180,E1 6906.703,E2 6906.703} C_VEL
LIN {X 0,Y 484.347,Z 648.599,A -85,B 0,C 180,E1 6909.054,E2 6909.054} C_VEL
LIN {X 0,Y 481.657,Z 672.943,A -85,B 0,C 180,E1 6911.918,E2 6911.918} C_VEL
LIN {X 0,Y 479.403,Z 693.841,A -85,B 0,C 180,E1 6915.367,E2 6915.367} C_VEL
LIN {X 0,Y 477.66,Z 710.26,A -85,B 0,C 180,E1 6919.323,E2 6919.323} C_VEL
LIN {X 0,Y 476.81,Z 721.308,A -85,B 0,C 180,E1 6923.621,E2 6923.621} C_VEL
LIN {X 0,Y 476.553,Z 725.32,A -85,B 0,C 180,E1 6926.359,E2 6926.359} C_VEL
LIN {X 0,Y 476.402,Z 727.183,A -85,B 0,C 180,E1 6930.002,E2 6930.002} C_VEL
LIN {X 0,Y 476.6,Z 724.116,A -85,B 0,C 180,E1 6934.557,E2 6934.557} C_VEL
LIN {X 0,Y 477.158,Z 715.954,A -85,B 0,C 180,E1 6938.67,E2 6938.67} C_VEL
LIN {X 0,Y 478.492,Z 701.908,A -85,B 0,C 180,E1 6942.798,E2 6942.798} C_VEL
LIN {X 0,Y 480.566,Z 683.064,A -85,B 0,C 180,E1 6946.474,E2 6946.474} C_VEL
LIN {X 0,Y 483.143,Z 659.513,A -85,B 0,C 180,E1 6949.685,E2 6949.685} C_VEL
LIN {X 0,Y 485.798,Z 633.11,A -85,B 0,C 180,E1 6952.249,E2 6952.249} C_VEL
LIN {X 0,Y 486.773,Z 616.014,A -85,B 0,C 180,E1 6953.522,E2 6953.522} C_VEL
LIN {X 0,Y 476.654,Z 586.316,A -85,B 0,C 180,E1 6955.926,E2 6955.926} C_VEL
LIN {X 0,Y 474.922,Z 580.66,A -85,B 0,C 180,E1 6956.359,E2 6956.359} C_VEL
LIN {X 0,Y 474.727,Z 580.66,A -85,B 0,C 180,E1 6962.834,E2 6962.834} C_VEL
LIN {X 0,Y 474.762,Z 580.66,A -85,B 0,C 180,E1 6967.297,E2 6967.297} C_VEL
LIN {X 0,Y 474.641,Z 580.66,A -85,B 0,C 180,E1 6972.798,E2 6972.798} C_VEL
LIN {X 0,Y 474.648,Z 580.66,A -85,B 0,C 180,E1 6977.937,E2 6977.937} C_VEL
LIN {X 0,Y 474.683,Z 580.66,A -85,B 0,C 180,E1 6984.956,E2 6984.956} C_VEL
LIN {X 0,Y 474.787,Z 580.66,A -85,B 0,C 180,E1 6991.418,E2 6991.418} C_VEL
LIN {X 0,Y 475.037,Z 580.66,A -85,B 0,C 180,E1 6997.564,E2 6997.564} C_VEL
LIN {X 0,Y 475.068,Z 580.66,A -85,B 0,C 180,E1 7003.327,E2 7003.327} C_VEL
LIN {X 0,Y 475.14,Z 580.66,A -85,B 0,C 180,E1 7008.973,E2 7008.973} C_VEL
LIN {X 0,Y 475.454,Z 580.66,A -85,B 0,C 180,E1 7014.513,E2 7014.513} C_VEL
LIN {X 0,Y 475.585,Z 580.66,A -85,B 0,C 180,E1 7019.995,E2 7019.995} C_VEL
LIN {X 0,Y 475.405,Z 580.66,A -85,B 0,C 180,E1 7025.477,E2 7025.477} C_VEL
LIN {X 0,Y 475.233,Z 580.66,A -85,B 0,C 180,E1 7031.015,E2 7031.015} C_VEL
LIN {X 0,Y 475.08,Z 580.66,A -85,B 0,C 180,E1 7037.042,E2 7037.042} C_VEL
LIN {X 0,Y 475.003,Z 580.66,A -85,B 0,C 180,E1 7042.482,E2 7042.482} C_VEL
LIN {X 0,Y 474.814,Z 580.66,A -85,B 0,C 180,E1 7048.569,E2 7048.569} C_VEL
LIN {X 0,Y 474.715,Z 580.66,A -85,B 0,C 180,E1 7055.029,E2 7055.029} C_VEL
LIN {X 0,Y 474.626,Z 580.66,A -85,B 0,C 180,E1 7062.051,E2 7062.051} C_VEL
LIN {X 0,Y 474.687,Z 580.66,A -85,B 0,C 180,E1 7067.946,E2 7067.946} C_VEL
LIN {X 0,Y 474.756,Z 580.66,A -85,B 0,C 180,E1 7072.861,E2 7072.861} C_VEL
LIN {X 0,Y 474.803,Z 580.66,A -85,B 0,C 180,E1 7076.281,E2 7076.281} C_VEL
LIN {X 0,Y 475.504,Z 583.332,A -85,B 0,C 180,E1 7076.874,E2 7076.874} C_VEL
LIN {X 0,Y 477.186,Z 592.911,A -85,B 0,C 180,E1 7077.371,E2 7077.371} C_VEL
LIN {X 0,Y 478.829,Z 611.799,A -85,B 0,C 180,E1 7077.814,E2 7077.814} C_VEL
LIN {X 0,Y 479.23,Z 612.95,A -85,B 0,C 180,E1 7077.859,E2 7077.859} C_VEL
LIN {X 0,Y 483.223,Z 623.525,A -85,B 0,C 180,E1 7078.291,E2 7078.291} C_VEL
LIN {X 0,Y 481.936,Z 666.333,A -85,B 0,C 180,E1 7079.186,E2 7079.186} C_VEL
LIN {X 0,Y 479.673,Z 703.868,A -85,B 0,C 180,E1 7080.651,E2 7080.651} C_VEL
LIN {X 0,Y 476.979,Z 740.419,A -85,B 0,C 180,E1 7082.866,E2 7082.866} C_VEL
LIN {X 0,Y 474.367,Z 772.768,A -85,B 0,C 180,E1 7085.61,E2 7085.61} C_VEL
LIN {X 0,Y 471.974,Z 801.152,A -85,B 0,C 180,E1 7088.847,E2 7088.847} C_VEL
LIN {X 0,Y 470.032,Z 826.354,A -85,B 0,C 180,E1 7092.739,E2 7092.739} C_VEL
LIN {X 0,Y 468.902,Z 844.601,A -85,B 0,C 180,E1 7096.575,E2 7096.575} C_VEL
LIN {X 0,Y 468.223,Z 858.331,A -85,B 0,C 180,E1 7100.694,E2 7100.694} C_VEL
LIN {X 0,Y 467.947,Z 865.957,A -85,B 0,C 180,E1 7104.428,E2 7104.428} C_VEL
LIN {X 0,Y 467.898,Z 869.507,A -85,B 0,C 180,E1 7108.144,E2 7108.144} C_VEL
LIN {X 0,Y 467.942,Z 869.509,A -85,B 0,C 180,E1 7111.852,E2 7111.852} C_VEL
LIN {X 0,Y 468.011,Z 864.437,A -85,B 0,C 180,E1 7116.5,E2 7116.5} C_VEL
LIN {X 0,Y 468.316,Z 854.789,A -85,B 0,C 180,E1 7120.539,E2 7120.539} C_VEL
LIN {X 0,Y 469.151,Z 839.952,A -85,B 0,C 180,E1 7124.52,E2 7124.52} C_VEL
LIN {X 0,Y 470.571,Z 819.239,A -85,B 0,C 180,E1 7128.483,E2 7128.483} C_VEL
LIN {X 0,Y 472.763,Z 791.913,A -85,B 0,C 180,E1 7132.313,E2 7132.313} C_VEL
LIN {X 0,Y 475.27,Z 761.208,A -85,B 0,C 180,E1 7135.469,E2 7135.469} C_VEL
LIN {X 0,Y 478.044,Z 726.738,A -85,B 0,C 180,E1 7138.065,E2 7138.065} C_VEL
LIN {X 0,Y 480.675,Z 689.451,A -85,B 0,C 180,E1 7139.993,E2 7139.993} C_VEL
LIN {X 0,Y 482.633,Z 652.595,A -85,B 0,C 180,E1 7141.171,E2 7141.171} C_VEL
LIN {X 0,Y 482.592,Z 620.644,A -85,B 0,C 180,E1 7141.797,E2 7141.797} C_VEL
LIN {X 0,Y 466.928,Z 580.66,A -85,B 0,C 180,E1 7143.628,E2 7143.628} C_VEL
LIN {X 0,Y 466.674,Z 580.66,A -85,B 0,C 180,E1 7150.453,E2 7150.453} C_VEL
LIN {X 0,Y 466.803,Z 580.66,A -85,B 0,C 180,E1 7157.076,E2 7157.076} C_VEL
LIN {X 0,Y 466.738,Z 580.66,A -85,B 0,C 180,E1 7161.958,E2 7161.958} C_VEL
LIN {X 0,Y 466.802,Z 580.66,A -85,B 0,C 180,E1 7168.745,E2 7168.745} C_VEL
LIN {X 0,Y 467.025,Z 580.66,A -85,B 0,C 180,E1 7175.187,E2 7175.187} C_VEL
LIN {X 0,Y 467.185,Z 580.66,A -85,B 0,C 180,E1 7181.096,E2 7181.096} C_VEL
LIN {X 0,Y 467.115,Z 580.66,A -85,B 0,C 180,E1 7186.891,E2 7186.891} C_VEL
LIN {X 0,Y 467.444,Z 580.66,A -85,B 0,C 180,E1 7192.561,E2 7192.561} C_VEL
LIN {X 0,Y 467.745,Z 580.66,A -85,B 0,C 180,E1 7198.15,E2 7198.15} C_VEL
LIN {X 0,Y 467.678,Z 580.66,A -85,B 0,C 180,E1 7203.717,E2 7203.717} C_VEL
LIN {X 0,Y 467.389,Z 580.66,A -85,B 0,C 180,E1 7209.326,E2 7209.326} C_VEL
LIN {X 0,Y 467.218,Z 580.66,A -85,B 0,C 180,E1 7215.03,E2 7215.03} C_VEL
LIN {X 0,Y 467.103,Z 580.66,A -85,B 0,C 180,E1 7220.894,E2 7220.894} C_VEL
LIN {X 0,Y 466.929,Z 580.66,A -85,B 0,C 180,E1 7227.003,E2 7227.003} C_VEL
LIN {X 0,Y 466.882,Z 580.66,A -85,B 0,C 180,E1 7233.461,E2 7233.461} C_VEL
LIN {X 0,Y 466.732,Z 580.66,A -85,B 0,C 180,E1 7238.877,E2 7238.877} C_VEL
LIN {X 0,Y 466.616,Z 580.66,A -85,B 0,C 180,E1 7245.555,E2 7245.555} C_VEL
LIN {X 0,Y 466.783,Z 580.66,A -85,B 0,C 180,E1 7251.958,E2 7251.958} C_VEL
LIN {X 0,Y 466.886,Z 580.66,A -85,B 0,C 180,E1 7258.747,E2 7258.747} C_VEL
LIN {X 0,Y 466.928,Z 580.984,A -85,B 0,C 180,E1 7263.038,E2 7263.038} C_VEL
LIN {X 0,Y 477.721,Z 612.12,A -85,B 0,C 180,E1 7265.493,E2 7265.493} C_VEL
LIN {X 0,Y 479.743,Z 621.597,A -85,B 0,C 180,E1 7266.312,E2 7266.312} C_VEL
LIN {X 0,Y 477.11,Z 650.09,A -85,B 0,C 180,E1 7268.72,E2 7268.72} C_VEL
LIN {X 0,Y 474.288,Z 674.328,A -85,B 0,C 180,E1 7271.627,E2 7271.627} C_VEL
LIN {X 0,Y 471.849,Z 695.162,A -85,B 0,C 180,E1 7275.128,E2 7275.128} C_VEL
LIN {X 0,Y 470.003,Z 711.536,A -85,B 0,C 180,E1 7279.147,E2 7279.147} C_VEL
LIN {X 0,Y 469.045,Z 722.535,A -85,B 0,C 180,E1 7283.515,E2 7283.515} C_VEL
LIN {X 0,Y 468.756,Z 726.522,A -85,B 0,C 180,E1 7286.298,E2 7286.298} C_VEL
LIN {X 0,Y 468.6,Z 728.369,A -85,B 0,C 180,E1 7290.002,E2 7290.002} C_VEL
LIN {X 0,Y 468.83,Z 725.322,A -85,B 0,C 180,E1 7294.632,E2 7294.632} C_VEL
LIN {X 0,Y 469.448,Z 717.207,A -85,B 0,C 180,E1 7298.814,E2 7298.814} C_VEL
LIN {X 0,Y 470.891,Z 703.218,A -85,B 0,C 180,E1 7303.008,E2 7303.008} C_VEL
LIN {X 0,Y 473.091,Z 684.423,A -85,B 0,C 180,E1 7306.741,E2 7306.741} C_VEL
LIN {X 0,Y 475.832,Z 660.961,A -85,B 0,C 180,E1 7310.001,E2 7310.001} C_VEL
LIN {X 0,Y 478.778,Z 633.398,A -85,B 0,C 180,E1 7312.702,E2 7312.702} C_VEL
LIN {X 0,Y 479.42,Z 617.643,A -85,B 0,C 180,E1 7313.916,E2 7313.916} C_VEL
LIN {X 0,Y 468.959,Z 587.057,A -85,B 0,C 180,E1 7316.453,E2 7316.453} C_VEL
LIN {X 0,Y 466.948,Z 580.66,A -85,B 0,C 180,E1 7316.998,E2 7316.998} C_VEL
LIN {X 0,Y 466.798,Z 580.66,A -85,B 0,C 180,E1 7323.464,E2 7323.464} C_VEL
LIN {X 0,Y 466.731,Z 580.66,A -85,B 0,C 180,E1 7330.452,E2 7330.452} C_VEL
LIN {X 0,Y 466.763,Z 580.66,A -85,B 0,C 180,E1 7337.058,E2 7337.058} C_VEL
LIN {X 0,Y 466.694,Z 580.66,A -85,B 0,C 180,E1 7341.94,E2 7341.94} C_VEL
LIN {X 0,Y 466.768,Z 580.66,A -85,B 0,C 180,E1 7348.73,E2 7348.73} C_VEL
LIN {X 0,Y 467.027,Z 580.66,A -85,B 0,C 180,E1 7355.195,E2 7355.195} C_VEL
LIN {X 0,Y 467.177,Z 580.66,A -85,B 0,C 180,E1 7361.085,E2 7361.085} C_VEL
LIN {X 0,Y 467.091,Z 580.66,A -85,B 0,C 180,E1 7366.88,E2 7366.88} C_VEL
LIN {X 0,Y 467.461,Z 580.66,A -85,B 0,C 180,E1 7372.551,E2 7372.551} C_VEL
LIN {X 0,Y 467.775,Z 580.66,A -85,B 0,C 180,E1 7378.14,E2 7378.14} C_VEL
LIN {X 0,Y 467.664,Z 580.66,A -85,B 0,C 180,E1 7383.707,E2 7383.707} C_VEL
LIN {X 0,Y 467.402,Z 580.66,A -85,B 0,C 180,E1 7389.316,E2 7389.316} C_VEL
LIN {X 0,Y 467.229,Z 580.66,A -85,B 0,C 180,E1 7395.019,E2 7395.019} C_VEL
LIN {X 0,Y 467.1,Z 580.66,A -85,B 0,C 180,E1 7400.883,E2 7400.883} C_VEL
LIN {X 0,Y 466.928,Z 580.66,A -85,B 0,C 180,E1 7406.992,E2 7406.992} C_VEL
LIN {X 0,Y 466.798,Z 580.66,A -85,B 0,C 180,E1 7413.456,E2 7413.456} C_VEL
LIN {X 0,Y 466.676,Z 580.66,A -85,B 0,C 180,E1 7420.449,E2 7420.449} C_VEL
LIN {X 0,Y 466.799,Z 580.66,A -85,B 0,C 180,E1 7427.067,E2 7427.067} C_VEL
LIN {X 0,Y 466.745,Z 580.66,A -85,B 0,C 180,E1 7431.95,E2 7431.95} C_VEL
LIN {X 0,Y 466.931,Z 580.66,A -85,B 0,C 180,E1 7436.406,E2 7436.406} C_VEL
LIN {X 0,Y 479.23,Z 612.95,A -85,B 0,C 180,E1 7437.859,E2 7437.859} C_VEL
LIN {X 0,Y 480.421,Z 621.323,A -85,B 0,C 180,E1 7438.074,E2 7438.074} C_VEL
LIN {X 0,Y 475.737,Z 648.052,A -85,B 0,C 180,E1 7438.307,E2 7438.307} C_VEL
LIN {X 0,Y 473.505,Z 686.305,A -85,B 0,C 180,E1 7439.504,E2 7439.504} C_VEL
LIN {X 0,Y 470.843,Z 723.678,A -85,B 0,C 180,E1 7441.435,E2 7441.435} C_VEL
LIN {X 0,Y 467.827,Z 759.004,A -85,B 0,C 180,E1 7444.092,E2 7444.092} C_VEL
LIN {X 0,Y 465.118,Z 789.677,A -85,B 0,C 180,E1 7447.26,E2 7447.26} C_VEL
LIN {X 0,Y 462.906,Z 815.989,A -85,B 0,C 180,E1 7450.907,E2 7450.907} C_VEL
LIN {X 0,Y 461.342,Z 837.949,A -85,B 0,C 180,E1 7455.091,E2 7455.091} C_VEL
LIN {X 0,Y 460.514,Z 852.953,A -85,B 0,C 180,E1 7459.101,E2 7459.101} C_VEL
LIN {X 0,Y 460.205,Z 863.421,A -85,B 0,C 180,E1 7463.386,E2 7463.386} C_VEL
LIN {X 0,Y 460.051,Z 867.444,A -85,B 0,C 180,E1 7466.224,E2 7466.224} C_VEL
LIN {X 0,Y 459.996,Z 869.432,A -85,B 0,C 180,E1 7469.998,E2 7469.998} C_VEL
LIN {X 0,Y 460.148,Z 866.379,A -85,B 0,C 180,E1 7474.717,E2 7474.717} C_VEL
LIN {X 0,Y 460.362,Z 857.81,A -85,B 0,C 180,E1 7479.174,E2 7479.174} C_VEL
LIN {X 0,Y 460.974,Z 844.644,A -85,B 0,C 180,E1 7483.29,E2 7483.29} C_VEL
LIN {X 0,Y 462.044,Z 827.046,A -85,B 0,C 180,E1 7487.15,E2 7487.15} C_VEL
LIN {X 0,Y 463.837,Z 804.658,A -85,B 0,C 180,E1 7490.79,E2 7490.79} C_VEL
LIN {X 0,Y 466.387,Z 775.689,A -85,B 0,C 180,E1 7494.305,E2 7494.305} C_VEL
LIN {X 0,Y 469.341,Z 742.16,A -85,B 0,C 180,E1 7497.285,E2 7497.285} C_VEL
LIN {X 0,Y 472.137,Z 706.675,A -85,B 0,C 180,E1 7499.539,E2 7499.539} C_VEL
LIN {X 0,Y 474.717,Z 667.701,A -85,B 0,C 180,E1 7501.171,E2 7501.171} C_VEL
LIN {X 0,Y 476.117,Z 625.733,A -85,B 0,C 180,E1 7502.111,E2 7502.111} C_VEL
LIN {X 0,Y 458.946,Z 580.66,A -85,B 0,C 180,E1 7504.194,E2 7504.194} C_VEL
LIN {X 0,Y 458.805,Z 580.66,A -85,B 0,C 180,E1 7511.296,E2 7511.296} C_VEL
LIN {X 0,Y 458.884,Z 580.66,A -85,B 0,C 180,E1 7516.538,E2 7516.538} C_VEL
LIN {X 0,Y 458.806,Z 580.66,A -85,B 0,C 180,E1 7522.368,E2 7522.368} C_VEL
LIN {X 0,Y 458.904,Z 580.66,A -85,B 0,C 180,E1 7529.066,E2 7529.066} C_VEL
LIN {X 0,Y 459.036,Z 580.66,A -85,B 0,C 180,E1 7534.616,E2 7534.616} C_VEL
LIN {X 0,Y 459.273,Z 580.66,A -85,B 0,C 180,E1 7540.758,E2 7540.758} C_VEL
LIN {X 0,Y 459.2,Z 580.66,A -85,B 0,C 180,E1 7546.661,E2 7546.661} C_VEL
LIN {X 0,Y 459.518,Z 580.66,A -85,B 0,C 180,E1 7552.432,E2 7552.432} C_VEL
LIN {X 0,Y 459.833,Z 580.66,A -85,B 0,C 180,E1 7558.118,E2 7558.118} C_VEL
LIN {X 0,Y 459.761,Z 580.66,A -85,B 0,C 180,E1 7563.782,E2 7563.782} C_VEL
LIN {X 0,Y 459.486,Z 580.66,A -85,B 0,C 180,E1 7569.488,E2 7569.488} C_VEL
LIN {X 0,Y 459.286,Z 580.66,A -85,B 0,C 180,E1 7575.296,E2 7575.296} C_VEL
LIN {X 0,Y 459.149,Z 580.66,A -85,B 0,C 180,E1 7581.273,E2 7581.273} C_VEL
LIN {X 0,Y 458.986,Z 580.66,A -85,B 0,C 180,E1 7587.51,E2 7587.51} C_VEL
LIN {X 0,Y 458.898,Z 580.66,A -85,B 0,C 180,E1 7594.123,E2 7594.123} C_VEL
LIN {X 0,Y 458.769,Z 580.66,A -85,B 0,C 180,E1 7600.623,E2 7600.623} C_VEL
LIN {X 0,Y 458.698,Z 580.66,A -85,B 0,C 180,E1 7606.573,E2 7606.573} C_VEL
LIN {X 0,Y 458.865,Z 580.66,A -85,B 0,C 180,E1 7612.37,E2 7612.37} C_VEL
LIN {X 0,Y 458.974,Z 580.66,A -85,B 0,C 180,E1 7619.066,E2 7619.066} C_VEL
LIN {X 0,Y 458.976,Z 581.191,A -85,B 0,C 180,E1 7622.44,E2 7622.44} C_VEL
LIN {X 0,Y 469.816,Z 611.975,A -85,B 0,C 180,E1 7624.912,E2 7624.912} C_VEL
LIN {X 0,Y 472.627,Z 623.902,A -85,B 0,C 180,E1 7625.987,E2 7625.987} C_VEL
LIN {X 0,Y 469.733,Z 652.637,A -85,B 0,C 180,E1 7628.494,E2 7628.494} C_VEL
LIN {X 0,Y 466.721,Z 677.334,A -85,B 0,C 180,E1 7631.563,E2 7631.563} C_VEL
LIN {X 0,Y 464.187,Z 697.567,A -85,B 0,C 180,E1 7635.118,E2 7635.118} C_VEL
LIN {X 0,Y 462.316,Z 712.999,A -85,B 0,C 180,E1 7639.027,E2 7639.027} C_VEL
LIN {X 0,Y 461.271,Z 723.751,A -85,B 0,C 180,E1 7643.405,E2 7643.405} C_VEL
LIN {X 0,Y 460.974,Z 727.716,A -85,B 0,C 180,E1 7646.235,E2 7646.235} C_VEL
LIN {X 0,Y 460.79,Z 729.555,A -85,B 0,C 180,E1 7650.002,E2 7650.002} C_VEL
LIN {X 0,Y 461.066,Z 726.519,A -85,B 0,C 180,E1 7654.711,E2 7654.711} C_VEL
LIN {X 0,Y 461.721,Z 718.445,A -85,B 0,C 180,E1 7658.962,E2 7658.962} C_VEL
LIN {X 0,Y 463.276,Z 704.505,A -85,B 0,C 180,E1 7663.226,E2 7663.226} C_VEL
LIN {X 0,Y 465.632,Z 685.753,A -85,B 0,C 180,E1 7667.018,E2 7667.018} C_VEL
LIN {X 0,Y 468.525,Z 662.566,A -85,B 0,C 180,E1 7670.302,E2 7670.302} C_VEL
LIN {X 0,Y 471.652,Z 634.96,A -85,B 0,C 180,E1 7673.065,E2 7673.065} C_VEL
LIN {X 0,Y 472.166,Z 619.594,A -85,B 0,C 180,E1 7674.288,E2 7674.288} C_VEL
LIN {X 0,Y 462.193,Z 589.877,A -85,B 0,C 180,E1 7676.828,E2 7676.828} C_VEL
LIN {X 0,Y 459.002,Z 580.66,A -85,B 0,C 180,E1 7677.505,E2 7677.505} C_VEL
LIN {X 0,Y 458.821,Z 580.66,A -85,B 0,C 180,E1 7684.407,E2 7684.407} C_VEL
LIN {X 0,Y 458.832,Z 580.66,A -85,B 0,C 180,E1 7690.621,E2 7690.621} C_VEL
LIN {X 0,Y 458.837,Z 580.66,A -85,B 0,C 180,E1 7696.549,E2 7696.549} C_VEL
LIN {X 0,Y 458.765,Z 580.66,A -85,B 0,C 180,E1 7702.38,E2 7702.38} C_VEL
LIN {X 0,Y 458.854,Z 580.66,A -85,B 0,C 180,E1 7709.084,E2 7709.084} C_VEL
LIN {X 0,Y 459.047,Z 580.66,A -85,B 0,C 180,E1 7714.605,E2 7714.605} C_VEL
LIN {X 0,Y 459.271,Z 580.66,A -85,B 0,C 180,E1 7720.746,E2 7720.746} C_VEL
LIN {X 0,Y 459.195,Z 580.66,A -85,B 0,C 180,E1 7726.65,E2 7726.65} C_VEL
LIN {X 0,Y 459.532,Z 580.66,A -85,B 0,C 180,E1 7732.422,E2 7732.422} C_VEL
LIN {X 0,Y 459.864,Z 580.66,A -85,B 0,C 180,E1 7738.108,E2 7738.108} C_VEL
LIN {X 0,Y 459.748,Z 580.66,A -85,B 0,C 180,E1 7743.771,E2 7743.771} C_VEL
LIN {X 0,Y 459.5,Z 580.66,A -85,B 0,C 180,E1 7749.477,E2 7749.477} C_VEL
LIN {X 0,Y 459.295,Z 580.66,A -85,B 0,C 180,E1 7755.285,E2 7755.285} C_VEL
LIN {X 0,Y 459.146,Z 580.66,A -85,B 0,C 180,E1 7761.262,E2 7761.262} C_VEL
LIN {X 0,Y 458.98,Z 580.66,A -85,B 0,C 180,E1 7767.498,E2 7767.498} C_VEL
LIN {X 0,Y 458.806,Z 580.66,A -85,B 0,C 180,E1 7774.118,E2 7774.118} C_VEL
LIN {X 0,Y 458.782,Z 580.66,A -85,B 0,C 180,E1 7780.62,E2 7780.62} C_VEL
LIN {X 0,Y 458.857,Z 580.66,A -85,B 0,C 180,E1 7786.536,E2 7786.536} C_VEL
LIN {X 0,Y 458.814,Z 580.66,A -85,B 0,C 180,E1 7792.361,E2 7792.361} C_VEL
LIN {X 0,Y 459.005,Z 581.371,A -85,B 0,C 180,E1 7795.891,E2 7795.891} C_VEL
LIN {X 0,Y 476.186,Z 624.904,A -85,B 0,C 180,E1 7797.878,E2 7797.878} C_VEL
LIN {X 0,Y 475.737,Z 648.052,A -85,B 0,C 180,E1 7798.307,E2 7798.307} C_VEL
LIN {X 0,Y 471.318,Z 664.936,A -85,B 0,C 180,E1 7798.533,E2 7798.533} C_VEL
LIN {X 0,Y 466.867,Z 679.436,A -85,B 0,C 180,E1 7798.82,E2 7798.82} C_VEL
LIN {X 0,Y 466.62,Z 681.511,A -85,B 0,C 180,E1 7798.899,E2 7798.899} C_VEL
LIN {X 0,Y 463.788,Z 718.79,A -85,B 0,C 180,E1 7800.794,E2 7800.794} C_VEL
LIN {X 0,Y 460.661,Z 754.086,A -85,B 0,C 180,E1 7803.395,E2 7803.395} C_VEL
LIN {X 0,Y 457.744,Z 785.683,A -85,B 0,C 180,E1 7806.613,E2 7806.613} C_VEL
LIN {X 0,Y 455.357,Z 812.756,A -85,B 0,C 180,E1 7810.325,E2 7810.325} C_VEL
LIN {X 0,Y 453.644,Z 835.166,A -85,B 0,C 180,E1 7814.513,E2 7814.513} C_VEL
LIN {X 0,Y 452.657,Z 851.635,A -85,B 0,C 180,E1 7818.91,E2 7818.91} C_VEL
LIN {X 0,Y 452.376,Z 862.189,A -85,B 0,C 180,E1 7823.271,E2 7823.271} C_VEL
LIN {X 0,Y 452.259,Z 866.247,A -85,B 0,C 180,E1 7826.159,E2 7826.159} C_VEL
LIN {X 0,Y 452.2,Z 868.248,A -85,B 0,C 180,E1 7829.998,E2 7829.998} C_VEL
LIN {X 0,Y 452.327,Z 865.165,A -85,B 0,C 180,E1 7834.798,E2 7834.798} C_VEL
LIN {X 0,Y 452.544,Z 856.534,A -85,B 0,C 180,E1 7839.334,E2 7839.334} C_VEL
LIN {X 0,Y 453.142,Z 843.272,A -85,B 0,C 180,E1 7843.524,E2 7843.524} C_VEL
LIN {X 0,Y 454.286,Z 825.518,A -85,B 0,C 180,E1 7847.453,E2 7847.453} C_VEL
LIN {X 0,Y 456.125,Z 802.87,A -85,B 0,C 180,E1 7851.158,E2 7851.158} C_VEL
LIN {X 0,Y 458.763,Z 774.475,A -85,B 0,C 180,E1 7854.644,E2 7854.644} C_VEL
LIN {X 0,Y 461.891,Z 741.127,A -85,B 0,C 180,E1 7857.656,E2 7857.656} C_VEL
LIN {X 0,Y 464.91,Z 705.803,A -85,B 0,C 180,E1 7859.956,E2 7859.956} C_VEL
LIN {X 0,Y 467.639,Z 667.474,A -85,B 0,C 180,E1 7861.603,E2 7861.603} C_VEL
LIN {X 0,Y 469.129,Z 627.4,A -85,B 0,C 180,E1 7862.537,E2 7862.537} C_VEL
LIN {X 0,Y 452.213,Z 584.796,A -85,B 0,C 180,E1 7864.554,E2 7864.554} C_VEL
LIN {X 0,Y 450.991,Z 580.66,A -85,B 0,C 180,E1 7864.797,E2 7864.797} C_VEL
LIN {X 0,Y 450.844,Z 580.66,A -85,B 0,C 180,E1 7869.645,E2 7869.645} C_VEL
LIN {X 0,Y 450.864,Z 580.66,A -85,B 0,C 180,E1 7875.162,E2 7875.162} C_VEL
LIN {X 0,Y 450.926,Z 580.66,A -85,B 0,C 180,E1 7880.553,E2 7880.553} C_VEL
LIN {X 0,Y 450.87,Z 580.66,A -85,B 0,C 180,E1 7887.084,E2 7887.084} C_VEL
LIN {X 0,Y 451.006,Z 580.66,A -85,B 0,C 180,E1 7891.973,E2 7891.973} C_VEL
LIN {X 0,Y 451.23,Z 580.66,A -85,B 0,C 180,E1 7898.346,E2 7898.346} C_VEL
LIN {X 0,Y 451.265,Z 580.66,A -85,B 0,C 180,E1 7904.436,E2 7904.436} C_VEL
LIN {X 0,Y 451.447,Z 580.66,A -85,B 0,C 180,E1 7910.352,E2 7910.352} C_VEL
LIN {X 0,Y 451.683,Z 580.66,A -85,B 0,C 180,E1 7916.161,E2 7916.161} C_VEL
LIN {X 0,Y 451.866,Z 580.66,A -85,B 0,C 180,E1 7921.925,E2 7921.925} C_VEL
LIN {X 0,Y 451.596,Z 580.66,A -85,B 0,C 180,E1 7927.712,E2 7927.712} C_VEL
LIN {X 0,Y 451.407,Z 580.66,A -85,B 0,C 180,E1 7933.584,E2 7933.584} C_VEL
LIN {X 0,Y 451.23,Z 580.66,A -85,B 0,C 180,E1 7940.039,E2 7940.039} C_VEL
LIN {X 0,Y 451.115,Z 580.66,A -85,B 0,C 180,E1 7945.874,E2 7945.874} C_VEL
LIN {X 0,Y 450.952,Z 580.66,A -85,B 0,C 180,E1 7952.932,E2 7952.932} C_VEL
LIN {X 0,Y 450.876,Z 580.66,A -85,B 0,C 180,E1 7959.439,E2 7959.439} C_VEL
LIN {X 0,Y 450.705,Z 580.66,A -85,B 0,C 180,E1 7965.138,E2 7965.138} C_VEL
LIN {X 0,Y 450.889,Z 580.66,A -85,B 0,C 180,E1 7970.57,E2 7970.57} C_VEL
LIN {X 0,Y 450.982,Z 580.66,A -85,B 0,C 180,E1 7977.076,E2 7977.076} C_VEL
LIN {X 0,Y 451.092,Z 581.191,A -85,B 0,C 180,E1 7981.815,E2 7981.815} C_VEL
LIN {X 0,Y 462.143,Z 612.658,A -85,B 0,C 180,E1 7984.386,E2 7984.386} C_VEL
LIN {X 0,Y 465.554,Z 625.496,A -85,B 0,C 180,E1 7985.599,E2 7985.599} C_VEL
LIN {X 0,Y 462.513,Z 654.05,A -85,B 0,C 180,E1 7988.141,E2 7988.141} C_VEL
LIN {X 0,Y 459.343,Z 678.676,A -85,B 0,C 180,E1 7991.256,E2 7991.256} C_VEL
LIN {X 0,Y 456.655,Z 698.844,A -85,B 0,C 180,E1 7994.867,E2 7994.867} C_VEL
LIN {X 0,Y 454.661,Z 714.24,A -85,B 0,C 180,E1 7998.84,E2 7998.84} C_VEL
LIN {X 0,Y 453.51,Z 724.958,A -85,B 0,C 180,E1 8003.292,E2 8003.292} C_VEL
LIN {X 0,Y 453.197,Z 728.907,A -85,B 0,C 180,E1 8006.171,E2 8006.171} C_VEL
LIN {X 0,Y 452.996,Z 730.739,A -85,B 0,C 180,E1 8010.002,E2 8010.002} C_VEL
LIN {X 0,Y 453.283,Z 727.716,A -85,B 0,C 180,E1 8014.792,E2 8014.792} C_VEL
LIN {X 0,Y 454.005,Z 719.671,A -85,B 0,C 180,E1 8019.116,E2 8019.116} C_VEL
LIN {X 0,Y 455.666,Z 705.777,A -85,B 0,C 180,E1 8023.451,E2 8023.451} C_VEL
LIN {X 0,Y 458.175,Z 687.066,A -85,B 0,C 180,E1 8027.303,E2 8027.303} C_VEL
LIN {X 0,Y 461.235,Z 663.961,A -85,B 0,C 180,E1 8030.638,E2 8030.638} C_VEL
LIN {X 0,Y 464.476,Z 636.962,A -85,B 0,C 180,E1 8033.4,E2 8033.4} C_VEL
LIN {X 0,Y 465.264,Z 622.856,A -85,B 0,C 180,E1 8034.537,E2 8034.537} C_VEL
LIN {X 0,Y 455.163,Z 592.333,A -85,B 0,C 180,E1 8037.253,E2 8037.253} C_VEL
LIN {X 0,Y 450.996,Z 580.66,A -85,B 0,C 180,E1 8038.179,E2 8038.179} C_VEL
LIN {X 0,Y 450.886,Z 580.66,A -85,B 0,C 180,E1 8044.811,E2 8044.811} C_VEL
LIN {X 0,Y 450.909,Z 580.66,A -85,B 0,C 180,E1 8049.642,E2 8049.642} C_VEL
LIN {X 0,Y 450.838,Z 580.66,A -85,B 0,C 180,E1 8055.144,E2 8055.144} C_VEL
LIN {X 0,Y 450.87,Z 580.66,A -85,B 0,C 180,E1 8060.567,E2 8060.567} C_VEL
LIN {X 0,Y 450.827,Z 580.66,A -85,B 0,C 180,E1 8067.099,E2 8067.099} C_VEL
LIN {X 0,Y 451.13,Z 580.66,A -85,B 0,C 180,E1 8074.127,E2 8074.127} C_VEL
LIN {X 0,Y 451.315,Z 580.66,A -85,B 0,C 180,E1 8080.393,E2 8080.393} C_VEL
LIN {X 0,Y 451.306,Z 580.66,A -85,B 0,C 180,E1 8086.633,E2 8086.633} C_VEL
LIN {X 0,Y 451.637,Z 580.66,A -85,B 0,C 180,E1 8092.288,E2 8092.288} C_VEL
LIN {X 0,Y 451.969,Z 580.66,A -85,B 0,C 180,E1 8098.075,E2 8098.075} C_VEL
LIN {X 0,Y 451.852,Z 580.66,A -85,B 0,C 180,E1 8103.837,E2 8103.837} C_VEL
LIN {X 0,Y 451.568,Z 580.66,A -85,B 0,C 180,E1 8109.645,E2 8109.645} C_VEL
LIN {X 0,Y 451.366,Z 580.66,A -85,B 0,C 180,E1 8115.56,E2 8115.56} C_VEL
LIN {X 0,Y 451.214,Z 580.66,A -85,B 0,C 180,E1 8121.654,E2 8121.654} C_VEL
LIN {X 0,Y 450.996,Z 580.66,A -85,B 0,C 180,E1 8128.028,E2 8128.028} C_VEL
LIN {X 0,Y 450.861,Z 580.66,A -85,B 0,C 180,E1 8134.805,E2 8134.805} C_VEL
LIN {X 0,Y 450.849,Z 580.66,A -85,B 0,C 180,E1 8139.64,E2 8139.64} C_VEL
LIN {X 0,Y 450.852,Z 580.66,A -85,B 0,C 180,E1 8145.151,E2 8145.151} C_VEL
LIN {X 0,Y 450.904,Z 580.66,A -85,B 0,C 180,E1 8150.551,E2 8150.551} C_VEL
LIN {X 0,Y 451.012,Z 580.868,A -85,B 0,C 180,E1 8155.28,E2 8155.28} C_VEL
LIN {X 0,Y 469.185,Z 626.581,A -85,B 0,C 180,E1 8157.452,E2 8157.452} C_VEL
LIN {X 0,Y 467.501,Z 668.691,A -85,B 0,C 180,E1 8158.431,E2 8158.431} C_VEL
LIN {X 0,Y 466.62,Z 681.511,A -85,B 0,C 180,E1 8158.899,E2 8158.899} C_VEL
LIN {X 0,Y 457.109,Z 711.796,A -85,B 0,C 180,E1 8159.984,E2 8159.984} C_VEL
LIN {X 0,Y 456.867,Z 713.74,A -85,B 0,C 180,E1 8160.101,E2 8160.101} C_VEL
LIN {X 0,Y 453.572,Z 749.122,A -85,B 0,C 180,E1 8162.677,E2 8162.677} C_VEL
LIN {X 0,Y 450.32,Z 782.466,A -85,B 0,C 180,E1 8166.04,E2 8166.04} C_VEL
LIN {X 0,Y 447.802,Z 809.476,A -85,B 0,C 180,E1 8169.722,E2 8169.722} C_VEL
LIN {X 0,Y 445.942,Z 832.544,A -85,B 0,C 180,E1 8173.985,E2 8173.985} C_VEL
LIN {X 0,Y 444.929,Z 848.837,A -85,B 0,C 180,E1 8178.217,E2 8178.217} C_VEL
LIN {X 0,Y 444.606,Z 859.083,A -85,B 0,C 180,E1 8182.169,E2 8182.169} C_VEL
LIN {X 0,Y 444.437,Z 865.043,A -85,B 0,C 180,E1 8186.091,E2 8186.091} C_VEL
LIN {X 0,Y 444.389,Z 867.061,A -85,B 0,C 180,E1 8189.998,E2 8189.998} C_VEL
LIN {X 0,Y 444.448,Z 865.046,A -85,B 0,C 180,E1 8193.905,E2 8193.905} C_VEL
LIN {X 0,Y 444.673,Z 857.676,A -85,B 0,C 180,E1 8198.486,E2 8198.486} C_VEL
LIN {X 0,Y 445.201,Z 843.762,A -85,B 0,C 180,E1 8203.269,E2 8203.269} C_VEL
LIN {X 0,Y 446.417,Z 825.242,A -85,B 0,C 180,E1 8207.515,E2 8207.515} C_VEL
LIN {X 0,Y 448.283,Z 802.835,A -85,B 0,C 180,E1 8211.287,E2 8211.287} C_VEL
LIN {X 0,Y 451.116,Z 773.789,A -85,B 0,C 180,E1 8214.939,E2 8214.939} C_VEL
LIN {X 0,Y 454.493,Z 740.183,A -85,B 0,C 180,E1 8218.058,E2 8218.058} C_VEL
LIN {X 0,Y 457.769,Z 704.611,A -85,B 0,C 180,E1 8220.416,E2 8220.416} C_VEL
LIN {X 0,Y 460.636,Z 667.204,A -85,B 0,C 180,E1 8222.054,E2 8222.054} C_VEL
LIN {X 0,Y 461.949,Z 628.165,A -85,B 0,C 180,E1 8223.012,E2 8223.012} C_VEL
LIN {X 0,Y 444.396,Z 585.068,A -85,B 0,C 180,E1 8225.158,E2 8225.158} C_VEL
LIN {X 0,Y 443.006,Z 580.66,A -85,B 0,C 180,E1 8225.435,E2 8225.435} C_VEL
LIN {X 0,Y 442.838,Z 580.66,A -85,B 0,C 180,E1 8231.23,E2 8231.23} C_VEL
LIN {X 0,Y 442.899,Z 580.66,A -85,B 0,C 180,E1 8236.875,E2 8236.875} C_VEL
LIN {X 0,Y 442.926,Z 580.66,A -85,B 0,C 180,E1 8242.034,E2 8242.034} C_VEL
LIN {X 0,Y 442.965,Z 580.66,A -85,B 0,C 180,E1 8248.699,E2 8248.699} C_VEL
LIN {X 0,Y 443.134,Z 580.66,A -85,B 0,C 180,E1 8253.636,E2 8253.636} C_VEL
LIN {X 0,Y 443.38,Z 580.66,A -85,B 0,C 180,E1 8260.039,E2 8260.039} C_VEL
LIN {X 0,Y 443.358,Z 580.66,A -85,B 0,C 180,E1 8266.176,E2 8266.176} C_VEL
LIN {X 0,Y 443.69,Z 580.66,A -85,B 0,C 180,E1 8272.16,E2 8272.16} C_VEL
LIN {X 0,Y 444.026,Z 580.66,A -85,B 0,C 180,E1 8278.051,E2 8278.051} C_VEL
LIN {X 0,Y 443.943,Z 580.66,A -85,B 0,C 180,E1 8283.917,E2 8283.917} C_VEL
LIN {X 0,Y 443.639,Z 580.66,A -85,B 0,C 180,E1 8289.83,E2 8289.83} C_VEL
LIN {X 0,Y 443.424,Z 580.66,A -85,B 0,C 180,E1 8295.858,E2 8295.858} C_VEL
LIN {X 0,Y 443.255,Z 580.66,A -85,B 0,C 180,E1 8302.075,E2 8302.075} C_VEL
LIN {X 0,Y 443.068,Z 580.66,A -85,B 0,C 180,E1 8308.587,E2 8308.587} C_VEL
LIN {X 0,Y 443.052,Z 580.66,A -85,B 0,C 180,E1 8315.523,E2 8315.523} C_VEL
LIN {X 0,Y 442.797,Z 580.66,A -85,B 0,C 180,E1 8321.219,E2 8321.219} C_VEL
LIN {X 0,Y 442.745,Z 580.66,A -85,B 0,C 180,E1 8326.851,E2 8326.851} C_VEL
LIN {X 0,Y 442.959,Z 580.66,A -85,B 0,C 180,E1 8332.033,E2 8332.033} C_VEL
LIN {X 0,Y 443.073,Z 580.66,A -85,B 0,C 180,E1 8336.859,E2 8336.859} C_VEL
LIN {X 0,Y 443.148,Z 580.885,A -85,B 0,C 180,E1 8341.147,E2 8341.147} C_VEL
LIN {X 0,Y 454.308,Z 612.623,A -85,B 0,C 180,E1 8343.782,E2 8343.782} C_VEL
LIN {X 0,Y 458.342,Z 628.793,A -85,B 0,C 180,E1 8345.327,E2 8345.327} C_VEL
LIN {X 0,Y 455.01,Z 657.638,A -85,B 0,C 180,E1 8348.019,E2 8348.019} C_VEL
LIN {X 0,Y 451.742,Z 681.585,A -85,B 0,C 180,E1 8351.183,E2 8351.183} C_VEL
LIN {X 0,Y 448.793,Z 702.343,A -85,B 0,C 180,E1 8355.096,E2 8355.096} C_VEL
LIN {X 0,Y 446.661,Z 717.791,A -85,B 0,C 180,E1 8359.449,E2 8359.449} C_VEL
LIN {X 0,Y 445.669,Z 727.697,A -85,B 0,C 180,E1 8364.152,E2 8364.152} C_VEL
LIN {X 0,Y 445.226,Z 731.439,A -85,B 0,C 180,E1 8368.053,E2 8368.053} C_VEL
LIN {X 0,Y 445.312,Z 731.38,A -85,B 0,C 180,E1 8371.95,E2 8371.95} C_VEL
LIN {X 0,Y 445.65,Z 727.562,A -85,B 0,C 180,E1 8375.852,E2 8375.852} C_VEL
LIN {X 0,Y 446.578,Z 718.557,A -85,B 0,C 180,E1 8380.19,E2 8380.19} C_VEL
LIN {X 0,Y 448.675,Z 703.017,A -85,B 0,C 180,E1 8384.662,E2 8384.662} C_VEL
LIN {X 0,Y 451.394,Z 684.002,A -85,B 0,C 180,E1 8388.329,E2 8388.329} C_VEL
LIN {X 0,Y 454.687,Z 660.087,A -85,B 0,C 180,E1 8391.616,E2 8391.616} C_VEL
LIN {X 0,Y 457.921,Z 632.752,A -85,B 0,C 180,E1 8394.261,E2 8394.261} C_VEL
LIN {X 0,Y 457.814,Z 623.985,A -85,B 0,C 180,E1 8395.006,E2 8395.006} C_VEL
LIN {X 0,Y 447.696,Z 593.414,A -85,B 0,C 180,E1 8397.797,E2 8397.797} C_VEL
LIN {X 0,Y 443.053,Z 580.66,A -85,B 0,C 180,E1 8398.858,E2 8398.858} C_VEL
LIN {X 0,Y 442.963,Z 580.66,A -85,B 0,C 180,E1 8405.527,E2 8405.527} C_VEL
LIN {X 0,Y 442.868,Z 580.66,A -85,B 0,C 180,E1 8411.218,E2 8411.218} C_VEL
LIN {X 0,Y 442.861,Z 580.66,A -85,B 0,C 180,E1 8416.855,E2 8416.855} C_VEL
LIN {X 0,Y 442.874,Z 580.66,A -85,B 0,C 180,E1 8422.015,E2 8422.015} C_VEL
LIN {X 0,Y 442.927,Z 580.66,A -85,B 0,C 180,E1 8428.714,E2 8428.714} C_VEL
LIN {X 0,Y 443.141,Z 580.66,A -85,B 0,C 180,E1 8433.625,E2 8433.625} C_VEL
LIN {X 0,Y 443.387,Z 580.66,A -85,B 0,C 180,E1 8440.028,E2 8440.028} C_VEL
LIN {X 0,Y 443.337,Z 580.66,A -85,B 0,C 180,E1 8446.164,E2 8446.164} C_VEL
LIN {X 0,Y 443.704,Z 580.66,A -85,B 0,C 180,E1 8452.15,E2 8452.15} C_VEL
LIN {X 0,Y 444.056,Z 580.66,A -85,B 0,C 180,E1 8458.041,E2 8458.041} C_VEL
LIN {X 0,Y 443.934,Z 580.66,A -85,B 0,C 180,E1 8463.906,E2 8463.906} C_VEL
LIN {X 0,Y 443.653,Z 580.66,A -85,B 0,C 180,E1 8469.819,E2 8469.819} C_VEL
LIN {X 0,Y 443.427,Z 580.66,A -85,B 0,C 180,E1 8475.846,E2 8475.846} C_VEL
LIN {X 0,Y 443.253,Z 580.66,A -85,B 0,C 180,E1 8482.063,E2 8482.063} C_VEL
LIN {X 0,Y 443.052,Z 580.66,A -85,B 0,C 180,E1 8488.576,E2 8488.576} C_VEL
LIN {X 0,Y 442.924,Z 580.66,A -85,B 0,C 180,E1 8495.521,E2 8495.521} C_VEL
LIN {X 0,Y 442.837,Z 580.66,A -85,B 0,C 180,E1 8501.219,E2 8501.219} C_VEL
LIN {X 0,Y 442.885,Z 580.66,A -85,B 0,C 180,E1 8506.864,E2 8506.864} C_VEL
LIN {X 0,Y 442.924,Z 580.66,A -85,B 0,C 180,E1 8512.025,E2 8512.025} C_VEL
LIN {X 0,Y 443.041,Z 580.66,A -85,B 0,C 180,E1 8514.62,E2 8514.62} C_VEL
LIN {X 0,Y 462.05,Z 628.346,A -85,B 0,C 180,E1 8516.999,E2 8516.999} C_VEL
LIN {X 0,Y 460.405,Z 669.143,A -85,B 0,C 180,E1 8518.008,E2 8518.008} C_VEL
LIN {X 0,Y 457.524,Z 706.214,A -85,B 0,C 180,E1 8519.668,E2 8519.668} C_VEL
LIN {X 0,Y 456.867,Z 713.74,A -85,B 0,C 180,E1 8520.101,E2 8520.101} C_VEL
LIN {X 0,Y 453.489,Z 725.517,A -85,B 0,C 180,E1 8520.74,E2 8520.74} C_VEL
LIN {X 0,Y 446.847,Z 742.287,A -85,B 0,C 180,E1 8521.757,E2 8521.757} C_VEL
LIN {X 0,Y 446.58,Z 744.083,A -85,B 0,C 180,E1 8521.909,E2 8521.909} C_VEL
LIN {X 0,Y 443.24,Z 775.867,A -85,B 0,C 180,E1 8525.044,E2 8525.044} C_VEL
LIN {X 0,Y 440.314,Z 805.07,A -85,B 0,C 180,E1 8528.919,E2 8528.919} C_VEL
LIN {X 0,Y 438.27,Z 828.64,A -85,B 0,C 180,E1 8533.181,E2 8533.181} C_VEL
LIN {X 0,Y 437.212,Z 845.8,A -85,B 0,C 180,E1 8537.499,E2 8537.499} C_VEL
LIN {X 0,Y 436.794,Z 857.823,A -85,B 0,C 180,E1 8542.029,E2 8542.029} C_VEL
LIN {X 0,Y 436.626,Z 863.84,A -85,B 0,C 180,E1 8546.021,E2 8546.021} C_VEL
LIN {X 0,Y 436.585,Z 865.876,A -85,B 0,C 180,E1 8549.998,E2 8549.998} C_VEL
LIN {X 0,Y 436.637,Z 863.846,A -85,B 0,C 180,E1 8553.975,E2 8553.975} C_VEL
LIN {X 0,Y 436.82,Z 856.402,A -85,B 0,C 180,E1 8558.64,E2 8558.64} C_VEL
LIN {X 0,Y 437.381,Z 842.343,A -85,B 0,C 180,E1 8563.51,E2 8563.51} C_VEL
LIN {X 0,Y 438.63,Z 823.66,A -85,B 0,C 180,E1 8567.837,E2 8567.837} C_VEL
LIN {X 0,Y 440.738,Z 800.373,A -85,B 0,C 180,E1 8571.778,E2 8571.778} C_VEL
LIN {X 0,Y 443.761,Z 770.908,A -85,B 0,C 180,E1 8575.519,E2 8575.519} C_VEL
LIN {X 0,Y 447.226,Z 738.259,A -85,B 0,C 180,E1 8578.565,E2 8578.565} C_VEL
LIN {X 0,Y 450.637,Z 703.801,A -85,B 0,C 180,E1 8580.876,E2 8580.876} C_VEL
LIN {X 0,Y 453.687,Z 666.464,A -85,B 0,C 180,E1 8582.537,E2 8582.537} C_VEL
LIN {X 0,Y 454.874,Z 629.891,A -85,B 0,C 180,E1 8583.482,E2 8583.482} C_VEL
LIN {X 0,Y 438.467,Z 589.385,A -85,B 0,C 180,E1 8585.55,E2 8585.55} C_VEL
LIN {X 0,Y 435.009,Z 580.66,A -85,B 0,C 180,E1 8586.068,E2 8586.068} C_VEL
LIN {X 0,Y 434.944,Z 580.66,A -85,B 0,C 180,E1 8593.038,E2 8593.038} C_VEL
LIN {X 0,Y 434.996,Z 580.66,A -85,B 0,C 180,E1 8598.608,E2 8598.608} C_VEL
LIN {X 0,Y 434.977,Z 580.66,A -85,B 0,C 180,E1 8603.728,E2 8603.728} C_VEL
LIN {X 0,Y 435.066,Z 580.66,A -85,B 0,C 180,E1 8610.454,E2 8610.454} C_VEL
LIN {X 0,Y 435.233,Z 580.66,A -85,B 0,C 180,E1 8615.333,E2 8615.333} C_VEL
LIN {X 0,Y 435.457,Z 580.66,A -85,B 0,C 180,E1 8621.771,E2 8621.771} C_VEL
LIN {X 0,Y 435.491,Z 580.66,A -85,B 0,C 180,E1 8627.966,E2 8627.966} C_VEL
LIN {X 0,Y 435.867,Z 580.66,A -85,B 0,C 180,E1 8634.024,E2 8634.024} C_VEL
LIN {X 0,Y 436.13,Z 580.66,A -85,B 0,C 180,E1 8640.006,E2 8640.006} C_VEL
LIN {X 0,Y 435.813,Z 580.66,A -85,B 0,C 180,E1 8645.988,E2 8645.988} C_VEL
LIN {X 0,Y 435.581,Z 580.66,A -85,B 0,C 180,E1 8652.043,E2 8652.043} C_VEL
LIN {X 0,Y 435.453,Z 580.66,A -85,B 0,C 180,E1 8658.241,E2 8658.241} C_VEL
LIN {X 0,Y 435.196,Z 580.66,A -85,B 0,C 180,E1 8665.245,E2 8665.245} C_VEL
LIN {X 0,Y 435.115,Z 580.66,A -85,B 0,C 180,E1 8671.469,E2 8671.469} C_VEL
LIN {X 0,Y 434.997,Z 580.66,A -85,B 0,C 180,E1 8676.823,E2 8676.823} C_VEL
LIN {X 0,Y 434.828,Z 580.66,A -85,B 0,C 180,E1 8683.016,E2 8683.016} C_VEL
LIN {X 0,Y 434.919,Z 580.66,A -85,B 0,C 180,E1 8689.992,E2 8689.992} C_VEL
LIN {X 0,Y 435.158,Z 580.66,A -85,B 0,C 180,E1 8696.628,E2 8696.628} C_VEL
LIN {X 0,Y 435.24,Z 581.271,A -85,B 0,C 180,E1 8700.483,E2 8700.483} C_VEL
LIN {X 0,Y 446.33,Z 611.932,A -85,B 0,C 180,E1 8703.103,E2 8703.103} C_VEL
LIN {X 0,Y 451.275,Z 630.76,A -85,B 0,C 180,E1 8704.951,E2 8704.951} C_VEL
LIN {X 0,Y 447.833,Z 659.015,A -85,B 0,C 180,E1 8707.647,E2 8707.647} C_VEL
LIN {X 0,Y 444.377,Z 682.881,A -85,B 0,C 180,E1 8710.859,E2 8710.859} C_VEL
LIN {X 0,Y 441.409,Z 702.487,A -85,B 0,C 180,E1 8714.586,E2 8714.586} C_VEL
LIN {X 0,Y 439.247,Z 717.337,A -85,B 0,C 180,E1 8718.668,E2 8718.668} C_VEL
LIN {X 0,Y 437.995,Z 727.363,A -85,B 0,C 180,E1 8723.053,E2 8723.053} C_VEL
LIN {X 0,Y 437.626,Z 731.287,A -85,B 0,C 180,E1 8726.034,E2 8726.034} C_VEL
LIN {X 0,Y 437.379,Z 733.112,A -85,B 0,C 180,E1 8730.002,E2 8730.002} C_VEL
LIN {X 0,Y 437.727,Z 730.103,A -85,B 0,C 180,E1 8734.962,E2 8734.962} C_VEL
LIN {X 0,Y 438.586,Z 722.106,A -85,B 0,C 180,E1 8739.439,E2 8739.439} C_VEL
LIN {X 0,Y 440.505,Z 708.285,A -85,B 0,C 180,E1 8743.923,E2 8743.923} C_VEL
LIN {X 0,Y 443.317,Z 689.651,A -85,B 0,C 180,E1 8747.903,E2 8747.903} C_VEL
LIN {X 0,Y 446.825,Z 666.005,A -85,B 0,C 180,E1 8751.426,E2 8751.426} C_VEL
LIN {X 0,Y 450.479,Z 638.128,A -85,B 0,C 180,E1 8754.341,E2 8754.341} C_VEL
LIN {X 0,Y 450.734,Z 626.639,A -85,B 0,C 180,E1 8755.337,E2 8755.337} C_VEL
LIN {X 0,Y 441.224,Z 597.018,A -85,B 0,C 180,E1 8758.148,E2 8758.148} C_VEL
LIN {X 0,Y 435.149,Z 580.66,A -85,B 0,C 180,E1 8759.55,E2 8759.55} C_VEL
LIN {X 0,Y 434.97,Z 580.66,A -85,B 0,C 180,E1 8766.282,E2 8766.282} C_VEL
LIN {X 0,Y 434.942,Z 580.66,A -85,B 0,C 180,E1 8773.021,E2 8773.021} C_VEL
LIN {X 0,Y 434.96,Z 580.66,A -85,B 0,C 180,E1 8778.589,E2 8778.589} C_VEL
LIN {X 0,Y 434.915,Z 580.66,A -85,B 0,C 180,E1 8783.708,E2 8783.708} C_VEL
LIN {X 0,Y 435.023,Z 580.66,A -85,B 0,C 180,E1 8788.524,E2 8788.524} C_VEL
LIN {X 0,Y 435.256,Z 580.66,A -85,B 0,C 180,E1 8795.322,E2 8795.322} C_VEL
LIN {X 0,Y 435.457,Z 580.66,A -85,B 0,C 180,E1 8801.759,E2 8801.759} C_VEL
LIN {X 0,Y 435.482,Z 580.66,A -85,B 0,C 180,E1 8807.954,E2 8807.954} C_VEL
LIN {X 0,Y 435.895,Z 580.66,A -85,B 0,C 180,E1 8814.013,E2 8814.013} C_VEL
LIN {X 0,Y 436.132,Z 580.66,A -85,B 0,C 180,E1 8819.994,E2 8819.994} C_VEL
LIN {X 0,Y 435.822,Z 580.66,A -85,B 0,C 180,E1 8825.977,E2 8825.977} C_VEL
LIN {X 0,Y 435.595,Z 580.66,A -85,B 0,C 180,E1 8832.031,E2 8832.031} C_VEL
LIN {X 0,Y 435.451,Z 580.66,A -85,B 0,C 180,E1 8838.23,E2 8838.23} C_VEL
LIN {X 0,Y 435.199,Z 580.66,A -85,B 0,C 180,E1 8845.237,E2 8845.237} C_VEL
LIN {X 0,Y 435.058,Z 580.66,A -85,B 0,C 180,E1 8851.461,E2 8851.461} C_VEL
LIN {X 0,Y 434.904,Z 580.66,A -85,B 0,C 180,E1 8856.801,E2 8856.801} C_VEL
LIN {X 0,Y 434.938,Z 580.66,A -85,B 0,C 180,E1 8863.026,E2 8863.026} C_VEL
LIN {X 0,Y 434.981,Z 580.66,A -85,B 0,C 180,E1 8868.597,E2 8868.597} C_VEL
LIN {X 0,Y 435.079,Z 580.869,A -85,B 0,C 180,E1 8873.998,E2 8873.998} C_VEL
LIN {X 0,Y 455.278,Z 630.9,A -85,B 0,C 180,E1 8876.569,E2 8876.569} C_VEL
LIN {X 0,Y 453.3,Z 670.12,A -85,B 0,C 180,E1 8877.589,E2 8877.589} C_VEL
LIN {X 0,Y 450.179,Z 707.672,A -85,B 0,C 180,E1 8879.338,E2 8879.338} C_VEL
LIN {X 0,Y 446.58,Z 744.083,A -85,B 0,C 180,E1 8881.909,E2 8881.909} C_VEL
LIN {X 0,Y 441.428,Z 758.377,A -85,B 0,C 180,E1 8883.046,E2 8883.046} C_VEL
LIN {X 0,Y 436.058,Z 771.912,A -85,B 0,C 180,E1 8884.316,E2 8884.316} C_VEL
LIN {X 0,Y 432.888,Z 800.976,A -85,B 0,C 180,E1 8888.147,E2 8888.147} C_VEL
LIN {X 0,Y 430.579,Z 825.902,A -85,B 0,C 180,E1 8892.608,E2 8892.608} C_VEL
LIN {X 0,Y 429.462,Z 842.713,A -85,B 0,C 180,E1 8896.751,E2 8896.751} C_VEL
LIN {X 0,Y 428.954,Z 855.091,A -85,B 0,C 180,E1 8901.184,E2 8901.184} C_VEL
LIN {X 0,Y 428.803,Z 862.636,A -85,B 0,C 180,E1 8905.949,E2 8905.949} C_VEL
LIN {X 0,Y 428.774,Z 864.689,A -85,B 0,C 180,E1 8909.998,E2 8909.998} C_VEL
LIN {X 0,Y 428.815,Z 862.636,A -85,B 0,C 180,E1 8914.047,E2 8914.047} C_VEL
LIN {X 0,Y 428.968,Z 855.057,A -85,B 0,C 180,E1 8918.828,E2 8918.828} C_VEL
LIN {X 0,Y 429.455,Z 842.713,A -85,B 0,C 180,E1 8923.245,E2 8923.245} C_VEL
LIN {X 0,Y 430.681,Z 824.713,A -85,B 0,C 180,E1 8927.648,E2 8927.648} C_VEL
LIN {X 0,Y 432.891,Z 800.957,A -85,B 0,C 180,E1 8931.855,E2 8931.855} C_VEL
LIN {X 0,Y 435.92,Z 772.894,A -85,B 0,C 180,E1 8935.572,E2 8935.572} C_VEL
LIN {X 0,Y 439.696,Z 739.755,A -85,B 0,C 180,E1 8938.818,E2 8938.818} C_VEL
LIN {X 0,Y 443.267,Z 705.772,A -85,B 0,C 180,E1 8941.195,E2 8941.195} C_VEL
LIN {X 0,Y 446.486,Z 669.209,A -85,B 0,C 180,E1 8942.91,E2 8942.91} C_VEL
LIN {X 0,Y 448.07,Z 632.264,A -85,B 0,C 180,E1 8943.935,E2 8943.935} C_VEL
LIN {X 0,Y 432.482,Z 593.492,A -85,B 0,C 180,E1 8945.964,E2 8945.964} C_VEL
LIN {X 0,Y 427.053,Z 580.66,A -85,B 0,C 180,E1 8946.713,E2 8946.713} C_VEL
LIN {X 0,Y 427.019,Z 580.66,A -85,B 0,C 180,E1 8952.347,E2 8952.347} C_VEL
LIN {X 0,Y 427.071,Z 580.66,A -85,B 0,C 180,E1 8958.111,E2 8958.111} C_VEL
LIN {X 0,Y 427.008,Z 580.66,A -85,B 0,C 180,E1 8964.633,E2 8964.633} C_VEL
LIN {X 0,Y 427.17,Z 580.66,A -85,B 0,C 180,E1 8970.257,E2 8970.257} C_VEL
LIN {X 0,Y 427.358,Z 580.66,A -85,B 0,C 180,E1 8977.084,E2 8977.084} C_VEL
LIN {X 0,Y 427.506,Z 580.66,A -85,B 0,C 180,E1 8983.547,E2 8983.547} C_VEL
LIN {X 0,Y 427.683,Z 580.66,A -85,B 0,C 180,E1 8989.81,E2 8989.81} C_VEL
LIN {X 0,Y 427.957,Z 580.66,A -85,B 0,C 180,E1 8995.948,E2 8995.948} C_VEL
LIN {X 0,Y 428.162,Z 580.66,A -85,B 0,C 180,E1 9002.032,E2 9002.032} C_VEL
LIN {X 0,Y 427.868,Z 580.66,A -85,B 0,C 180,E1 9008.143,E2 9008.143} C_VEL
LIN {X 0,Y 427.608,Z 580.66,A -85,B 0,C 180,E1 9014.356,E2 9014.356} C_VEL
LIN {X 0,Y 427.427,Z 580.66,A -85,B 0,C 180,E1 9020.752,E2 9020.752} C_VEL
LIN {X 0,Y 427.213,Z 580.66,A -85,B 0,C 180,E1 9027.631,E2 9027.631} C_VEL
LIN {X 0,Y 427.179,Z 580.66,A -85,B 0,C 180,E1 9032.123,E2 9032.123} C_VEL
LIN {X 0,Y 427.041,Z 580.66,A -85,B 0,C 180,E1 9038.744,E2 9038.744} C_VEL
LIN {X 0,Y 426.902,Z 580.66,A -85,B 0,C 180,E1 9045.187,E2 9045.187} C_VEL
LIN {X 0,Y 427.056,Z 580.66,A -85,B 0,C 180,E1 9051.266,E2 9051.266} C_VEL
LIN {X 0,Y 427.221,Z 580.66,A -85,B 0,C 180,E1 9058.281,E2 9058.281} C_VEL
LIN {X 0,Y 427.258,Z 581.177,A -85,B 0,C 180,E1 9059.761,E2 9059.761} C_VEL
LIN {X 0,Y 438.756,Z 612.582,A -85,B 0,C 180,E1 9062.521,E2 9062.521} C_VEL
LIN {X 0,Y 444.166,Z 633.28,A -85,B 0,C 180,E1 9064.617,E2 9064.617} C_VEL
LIN {X 0,Y 440.49,Z 661.484,A -85,B 0,C 180,E1 9067.388,E2 9067.388} C_VEL
LIN {X 0,Y 436.782,Z 685.668,A -85,B 0,C 180,E1 9070.776,E2 9070.776} C_VEL
LIN {X 0,Y 433.526,Z 705.902,A -85,B 0,C 180,E1 9074.818,E2 9074.818} C_VEL
LIN {X 0,Y 431.346,Z 719.964,A -85,B 0,C 180,E1 9078.974,E2 9078.974} C_VEL
LIN {X 0,Y 430.23,Z 728.564,A -85,B 0,C 180,E1 9082.927,E2 9082.927} C_VEL
LIN {X 0,Y 429.846,Z 732.476,A -85,B 0,C 180,E1 9085.962,E2 9085.962} C_VEL
LIN {X 0,Y 429.569,Z 734.298,A -85,B 0,C 180,E1 9090.002,E2 9090.002} C_VEL
LIN {X 0,Y 429.94,Z 731.297,A -85,B 0,C 180,E1 9095.053,E2 9095.053} C_VEL
LIN {X 0,Y 430.891,Z 723.317,A -85,B 0,C 180,E1 9099.61,E2 9099.61} C_VEL
LIN {X 0,Y 432.927,Z 709.531,A -85,B 0,C 180,E1 9104.172,E2 9104.172} C_VEL
LIN {X 0,Y 435.903,Z 690.93,A -85,B 0,C 180,E1 9108.218,E2 9108.218} C_VEL
LIN {X 0,Y 439.618,Z 667.26,A -85,B 0,C 180,E1 9111.808,E2 9111.808} C_VEL
LIN {X 0,Y 443.421,Z 639.61,A -85,B 0,C 180,E1 9114.755,E2 9114.755} C_VEL
LIN {X 0,Y 443.797,Z 629.543,A -85,B 0,C 180,E1 9115.646,E2 9115.646} C_VEL
LIN {X 0,Y 434.86,Z 600.997,A -85,B 0,C 180,E1 9118.458,E2 9118.458} C_VEL
LIN {X 0,Y 427.162,Z 580.66,A -85,B 0,C 180,E1 9120.236,E2 9120.236} C_VEL
LIN {X 0,Y 427.026,Z 580.66,A -85,B 0,C 180,E1 9127.068,E2 9127.068} C_VEL
LIN {X 0,Y 427.013,Z 580.66,A -85,B 0,C 180,E1 9132.353,E2 9132.353} C_VEL
LIN {X 0,Y 427.025,Z 580.66,A -85,B 0,C 180,E1 9138.124,E2 9138.124} C_VEL
LIN {X 0,Y 426.951,Z 580.66,A -85,B 0,C 180,E1 9144.651,E2 9144.651} C_VEL
LIN {X 0,Y 427.139,Z 580.66,A -85,B 0,C 180,E1 9150.242,E2 9150.242} C_VEL
LIN {X 0,Y 427.384,Z 580.66,A -85,B 0,C 180,E1 9157.086,E2 9157.086} C_VEL
LIN {X 0,Y 427.501,Z 580.66,A -85,B 0,C 180,E1 9163.535,E2 9163.535} C_VEL
LIN {X 0,Y 427.658,Z 580.66,A -85,B 0,C 180,E1 9169.798,E2 9169.798} C_VEL
LIN {X 0,Y 427.989,Z 580.66,A -85,B 0,C 180,E1 9175.937,E2 9175.937} C_VEL
LIN {X 0,Y 428.101,Z 580.66,A -85,B 0,C 180,E1 9182.021,E2 9182.021} C_VEL
LIN {X 0,Y 427.878,Z 580.66,A -85,B 0,C 180,E1 9188.131,E2 9188.131} C_VEL
LIN {X 0,Y 427.614,Z 580.66,A -85,B 0,C 180,E1 9194.344,E2 9194.344} C_VEL
LIN {X 0,Y 427.443,Z 580.66,A -85,B 0,C 180,E1 9200.739,E2 9200.739} C_VEL
LIN {X 0,Y 427.204,Z 580.66,A -85,B 0,C 180,E1 9207.621,E2 9207.621} C_VEL
LIN {X 0,Y 427.123,Z 580.66,A -85,B 0,C 180,E1 9212.114,E2 9212.114} C_VEL
LIN {X 0,Y 427,Z 580.66,A -85,B 0,C 180,E1 9218.731,E2 9218.731} C_VEL
LIN {X 0,Y 427.052,Z 580.66,A -85,B 0,C 180,E1 9225.15,E2 9225.15} C_VEL
LIN {X 0,Y 427.047,Z 580.66,A -85,B 0,C 180,E1 9231.249,E2 9231.249} C_VEL
LIN {X 0,Y 427.11,Z 580.66,A -85,B 0,C 180,E1 9233.284,E2 9233.284} C_VEL
LIN {X 0,Y 445.88,Z 626.418,A -85,B 0,C 180,E1 9235.786,E2 9235.786} C_VEL
LIN {X 0,Y 448.443,Z 634.284,A -85,B 0,C 180,E1 9236.142,E2 9236.142} C_VEL
LIN {X 0,Y 446.087,Z 672.913,A -85,B 0,C 180,E1 9237.223,E2 9237.223} C_VEL
LIN {X 0,Y 442.806,Z 709.684,A -85,B 0,C 180,E1 9239.027,E2 9239.027} C_VEL
LIN {X 0,Y 439.042,Z 745.118,A -85,B 0,C 180,E1 9241.643,E2 9241.643} C_VEL
LIN {X 0,Y 436.058,Z 771.912,A -85,B 0,C 180,E1 9244.316,E2 9244.316} C_VEL
LIN {X 0,Y 430.68,Z 784.758,A -85,B 0,C 180,E1 9245.74,E2 9245.74} C_VEL
LIN {X 0,Y 425.53,Z 796.696,A -85,B 0,C 180,E1 9247.306,E2 9247.306} C_VEL
LIN {X 0,Y 423.083,Z 820.651,A -85,B 0,C 180,E1 9251.49,E2 9251.49} C_VEL
LIN {X 0,Y 421.703,Z 840.244,A -85,B 0,C 180,E1 9256.18,E2 9256.18} C_VEL
LIN {X 0,Y 421.142,Z 853.812,A -85,B 0,C 180,E1 9261.019,E2 9261.019} C_VEL
LIN {X 0,Y 421,Z 861.429,A -85,B 0,C 180,E1 9265.874,E2 9265.874} C_VEL
LIN {X 0,Y 420.979,Z 863.505,A -85,B 0,C 180,E1 9269.998,E2 9269.998} C_VEL
LIN {X 0,Y 421.012,Z 861.429,A -85,B 0,C 180,E1 9274.123,E2 9274.123} C_VEL
LIN {X 0,Y 421.152,Z 853.777,A -85,B 0,C 180,E1 9278.994,E2 9278.994} C_VEL
LIN {X 0,Y 421.716,Z 840.144,A -85,B 0,C 180,E1 9283.846,E2 9283.846} C_VEL
LIN {X 0,Y 423.149,Z 820.664,A -85,B 0,C 180,E1 9288.506,E2 9288.506} C_VEL
LIN {X 0,Y 425.569,Z 796.185,A -85,B 0,C 180,E1 9292.773,E2 9292.773} C_VEL
LIN {X 0,Y 429.017,Z 766.823,A -85,B 0,C 180,E1 9296.566,E2 9296.566} C_VEL
LIN {X 0,Y 433.015,Z 733.243,A -85,B 0,C 180,E1 9299.738,E2 9299.738} C_VEL
LIN {X 0,Y 437.057,Z 697.237,A -85,B 0,C 180,E1 9302.129,E2 9302.129} C_VEL
LIN {X 0,Y 440.23,Z 660.194,A -85,B 0,C 180,E1 9303.71,E2 9303.71} C_VEL
LIN {X 0,Y 441.051,Z 634.023,A -85,B 0,C 180,E1 9304.428,E2 9304.428} C_VEL
LIN {X 0,Y 426.645,Z 597.843,A -85,B 0,C 180,E1 9306.374,E2 9306.374} C_VEL
LIN {X 0,Y 419.078,Z 580.66,A -85,B 0,C 180,E1 9307.447,E2 9307.447} C_VEL
LIN {X 0,Y 419.038,Z 580.66,A -85,B 0,C 180,E1 9313.737,E2 9313.737} C_VEL
LIN {X 0,Y 419.085,Z 580.66,A -85,B 0,C 180,E1 9319.444,E2 9319.444} C_VEL
LIN {X 0,Y 419.091,Z 580.66,A -85,B 0,C 180,E1 9326.188,E2 9326.188} C_VEL
LIN {X 0,Y 419.267,Z 580.66,A -85,B 0,C 180,E1 9332.008,E2 9332.008} C_VEL
LIN {X 0,Y 419.518,Z 580.66,A -85,B 0,C 180,E1 9338.851,E2 9338.851} C_VEL
LIN {X 0,Y 419.593,Z 580.66,A -85,B 0,C 180,E1 9345.376,E2 9345.376} C_VEL
LIN {X 0,Y 419.923,Z 580.66,A -85,B 0,C 180,E1 9351.714,E2 9351.714} C_VEL
LIN {X 0,Y 420.314,Z 580.66,A -85,B 0,C 180,E1 9357.941,E2 9357.941} C_VEL
LIN {X 0,Y 420.184,Z 580.66,A -85,B 0,C 180,E1 9364.138,E2 9364.138} C_VEL
LIN {X 0,Y 419.834,Z 580.66,A -85,B 0,C 180,E1 9370.394,E2 9370.394} C_VEL
LIN {X 0,Y 419.682,Z 580.66,A -85,B 0,C 180,E1 9376.78,E2 9376.78} C_VEL
LIN {X 0,Y 419.402,Z 580.66,A -85,B 0,C 180,E1 9383.403,E2 9383.403} C_VEL
LIN {X 0,Y 419.245,Z 580.66,A -85,B 0,C 180,E1 9390.377,E2 9390.377} C_VEL
LIN {X 0,Y 419.14,Z 580.66,A -85,B 0,C 180,E1 9397.378,E2 9397.378} C_VEL
LIN {X 0,Y 418.916,Z 580.66,A -85,B 0,C 180,E1 9403.714,E2 9403.714} C_VEL
LIN {X 0,Y 419.034,Z 580.66,A -85,B 0,C 180,E1 9409.434,E2 9409.434} C_VEL
LIN {X 0,Y 419.181,Z 580.66,A -85,B 0,C 180,E1 9416.184,E2 9416.184} C_VEL
LIN {X 0,Y 419.34,Z 580.764,A -85,B 0,C 180,E1 9419.006,E2 9419.006} C_VEL
LIN {X 0,Y 430.844,Z 612.08,A -85,B 0,C 180,E1 9421.805,E2 9421.805} C_VEL
LIN {X 0,Y 437.038,Z 635.743,A -85,B 0,C 180,E1 9424.265,E2 9424.265} C_VEL
LIN {X 0,Y 433.2,Z 663.922,A -85,B 0,C 180,E1 9427.121,E2 9427.121} C_VEL
LIN {X 0,Y 429.441,Z 686.947,A -85,B 0,C 180,E1 9430.434,E2 9430.434} C_VEL
LIN {X 0,Y 425.984,Z 707.139,A -85,B 0,C 180,E1 9434.542,E2 9434.542} C_VEL
LIN {X 0,Y 423.72,Z 720.897,A -85,B 0,C 180,E1 9438.668,E2 9438.668} C_VEL
LIN {X 0,Y 422.496,Z 729.759,A -85,B 0,C 180,E1 9442.797,E2 9442.797} C_VEL
LIN {X 0,Y 422.064,Z 733.664,A -85,B 0,C 180,E1 9445.888,E2 9445.888} C_VEL
LIN {X 0,Y 421.769,Z 735.483,A -85,B 0,C 180,E1 9450.002,E2 9450.002} C_VEL
LIN {X 0,Y 422.155,Z 732.489,A -85,B 0,C 180,E1 9455.146,E2 9455.146} C_VEL
LIN {X 0,Y 423.182,Z 724.541,A -85,B 0,C 180,E1 9459.781,E2 9459.781} C_VEL
LIN {X 0,Y 425.358,Z 710.771,A -85,B 0,C 180,E1 9464.43,E2 9464.43} C_VEL
LIN {X 0,Y 428.522,Z 692.199,A -85,B 0,C 180,E1 9468.543,E2 9468.543} C_VEL
LIN {X 0,Y 432.446,Z 668.401,A -85,B 0,C 180,E1 9472.216,E2 9472.216} C_VEL
LIN {X 0,Y 436.39,Z 641.135,A -85,B 0,C 180,E1 9475.173,E2 9475.173} C_VEL
LIN {X 0,Y 436.755,Z 632.171,A -85,B 0,C 180,E1 9475.997,E2 9475.997} C_VEL
LIN {X 0,Y 427.797,Z 603.04,A -85,B 0,C 180,E1 9478.958,E2 9478.958} C_VEL
LIN {X 0,Y 419.26,Z 580.66,A -85,B 0,C 180,E1 9480.988,E2 9480.988} C_VEL
LIN {X 0,Y 419.113,Z 580.66,A -85,B 0,C 180,E1 9487.89,E2 9487.89} C_VEL
LIN {X 0,Y 419.026,Z 580.66,A -85,B 0,C 180,E1 9493.719,E2 9493.719} C_VEL
LIN {X 0,Y 419.048,Z 580.66,A -85,B 0,C 180,E1 9499.425,E2 9499.425} C_VEL
LIN {X 0,Y 419.044,Z 580.66,A -85,B 0,C 180,E1 9506.205,E2 9506.205} C_VEL
LIN {X 0,Y 419.258,Z 580.66,A -85,B 0,C 180,E1 9511.994,E2 9511.994} C_VEL
LIN {X 0,Y 419.536,Z 580.66,A -85,B 0,C 180,E1 9518.84,E2 9518.84} C_VEL
LIN {X 0,Y 419.571,Z 580.66,A -85,B 0,C 180,E1 9525.363,E2 9525.363} C_VEL
LIN {X 0,Y 419.941,Z 580.66,A -85,B 0,C 180,E1 9531.702,E2 9531.702} C_VEL
LIN {X 0,Y 420.345,Z 580.66,A -85,B 0,C 180,E1 9537.93,E2 9537.93} C_VEL
LIN {X 0,Y 420.179,Z 580.66,A -85,B 0,C 180,E1 9544.127,E2 9544.127} C_VEL
LIN {X 0,Y 419.848,Z 580.66,A -85,B 0,C 180,E1 9550.382,E2 9550.382} C_VEL
LIN {X 0,Y 419.686,Z 580.66,A -85,B 0,C 180,E1 9556.768,E2 9556.768} C_VEL
LIN {X 0,Y 419.415,Z 580.66,A -85,B 0,C 180,E1 9563.39,E2 9563.39} C_VEL
LIN {X 0,Y 419.21,Z 580.66,A -85,B 0,C 180,E1 9570.366,E2 9570.366} C_VEL
LIN {X 0,Y 419.069,Z 580.66,A -85,B 0,C 180,E1 9577.359,E2 9577.359} C_VEL
LIN {X 0,Y 419.025,Z 580.66,A -85,B 0,C 180,E1 9583.725,E2 9583.725} C_VEL
LIN {X 0,Y 419.074,Z 580.66,A -85,B 0,C 180,E1 9589.433,E2 9589.433} C_VEL
LIN {X 0,Y 419.124,Z 580.66,A -85,B 0,C 180,E1 9592.546,E2 9592.546} C_VEL
LIN {X 0,Y 438.059,Z 625.639,A -85,B 0,C 180,E1 9595.16,E2 9595.16} C_VEL
LIN {X 0,Y 441.502,Z 637.473,A -85,B 0,C 180,E1 9595.691,E2 9595.691} C_VEL
LIN {X 0,Y 438.766,Z 677.202,A -85,B 0,C 180,E1 9596.907,E2 9596.907} C_VEL
LIN {X 0,Y 435.199,Z 713.442,A -85,B 0,C 180,E1 9598.834,E2 9598.834} C_VEL
LIN {X 0,Y 431.294,Z 748.007,A -85,B 0,C 180,E1 9601.529,E2 9601.529} C_VEL
LIN {X 0,Y 427.484,Z 779.892,A -85,B 0,C 180,E1 9604.987,E2 9604.987} C_VEL
LIN {X 0,Y 425.53,Z 796.696,A -85,B 0,C 180,E1 9607.306,E2 9607.306} C_VEL
LIN {X 0,Y 420.395,Z 807.836,A -85,B 0,C 180,E1 9609.019,E2 9609.019} C_VEL
LIN {X 0,Y 415.466,Z 817.95,A -85,B 0,C 180,E1 9610.864,E2 9610.864} C_VEL
LIN {X 0,Y 414.03,Z 836.225,A -85,B 0,C 180,E1 9615.167,E2 9615.167} C_VEL
LIN {X 0,Y 413.316,Z 850.542,A -85,B 0,C 180,E1 9619.978,E2 9619.978} C_VEL
LIN {X 0,Y 413.184,Z 859.064,A -85,B 0,C 180,E1 9624.742,E2 9624.742} C_VEL
LIN {X 0,Y 413.124,Z 861.749,A -85,B 0,C 180,E1 9627.898,E2 9627.898} C_VEL
LIN {X 0,Y 413.152,Z 861.756,A -85,B 0,C 180,E1 9632.098,E2 9632.098} C_VEL
LIN {X 0,Y 413.173,Z 857.698,A -85,B 0,C 180,E1 9636.309,E2 9636.309} C_VEL
LIN {X 0,Y 413.404,Z 847.932,A -85,B 0,C 180,E1 9641.083,E2 9641.083} C_VEL
LIN {X 0,Y 414.389,Z 832.21,A -85,B 0,C 180,E1 9645.902,E2 9645.902} C_VEL
LIN {X 0,Y 416.274,Z 810.941,A -85,B 0,C 180,E1 9650.489,E2 9650.489} C_VEL
LIN {X 0,Y 419.421,Z 783.587,A -85,B 0,C 180,E1 9654.81,E2 9654.81} C_VEL
LIN {X 0,Y 423.211,Z 753.816,A -85,B 0,C 180,E1 9658.278,E2 9658.278} C_VEL
LIN {X 0,Y 427.285,Z 719.504,A -85,B 0,C 180,E1 9661.21,E2 9661.21} C_VEL
LIN {X 0,Y 431.311,Z 682.877,A -85,B 0,C 180,E1 9663.335,E2 9663.335} C_VEL
LIN {X 0,Y 434.463,Z 644.597,A -85,B 0,C 180,E1 9664.672,E2 9664.672} C_VEL
LIN {X 0,Y 433.94,Z 635.414,A -85,B 0,C 180,E1 9664.957,E2 9664.957} C_VEL
LIN {X 0,Y 420.04,Z 600.498,A -85,B 0,C 180,E1 9666.904,E2 9666.904} C_VEL
LIN {X 0,Y 411.104,Z 580.66,A -85,B 0,C 180,E1 9668.259,E2 9668.259} C_VEL
LIN {X 0,Y 411.096,Z 580.66,A -85,B 0,C 180,E1 9675.601,E2 9675.601} C_VEL
LIN {X 0,Y 411.101,Z 580.66,A -85,B 0,C 180,E1 9681.246,E2 9681.246} C_VEL
LIN {X 0,Y 411.181,Z 580.66,A -85,B 0,C 180,E1 9687.871,E2 9687.871} C_VEL
LIN {X 0,Y 411.371,Z 580.66,A -85,B 0,C 180,E1 9693.797,E2 9693.797} C_VEL
LIN {X 0,Y 411.653,Z 580.66,A -85,B 0,C 180,E1 9700.676,E2 9700.676} C_VEL
LIN {X 0,Y 411.726,Z 580.66,A -85,B 0,C 180,E1 9707.26,E2 9707.26} C_VEL
LIN {X 0,Y 412.121,Z 580.66,A -85,B 0,C 180,E1 9713.678,E2 9713.678} C_VEL
LIN {X 0,Y 412.427,Z 580.66,A -85,B 0,C 180,E1 9720.006,E2 9720.006} C_VEL
LIN {X 0,Y 412.081,Z 580.66,A -85,B 0,C 180,E1 9726.334,E2 9726.334} C_VEL
LIN {X 0,Y 411.825,Z 580.66,A -85,B 0,C 180,E1 9732.749,E2 9732.749} C_VEL
LIN {X 0,Y 411.64,Z 580.66,A -85,B 0,C 180,E1 9739.337,E2 9739.337} C_VEL
LIN {X 0,Y 411.369,Z 580.66,A -85,B 0,C 180,E1 9746.216,E2 9746.216} C_VEL
LIN {X 0,Y 411.265,Z 580.66,A -85,B 0,C 180,E1 9753.526,E2 9753.526} C_VEL
LIN {X 0,Y 411.076,Z 580.66,A -85,B 0,C 180,E1 9759.339,E2 9759.339} C_VEL
LIN {X 0,Y 410.962,Z 580.66,A -85,B 0,C 180,E1 9765.578,E2 9765.578} C_VEL
LIN {X 0,Y 411.1,Z 580.66,A -85,B 0,C 180,E1 9771.241,E2 9771.241} C_VEL
LIN {X 0,Y 411.364,Z 580.66,A -85,B 0,C 180,E1 9778.213,E2 9778.213} C_VEL
LIN {X 0,Y 423.37,Z 612.911,A -85,B 0,C 180,E1 9781.193,E2 9781.193} C_VEL
LIN {X 0,Y 430.057,Z 637.199,A -85,B 0,C 180,E1 9783.816,E2 9783.816} C_VEL
LIN {X 0,Y 426.041,Z 665.258,A -85,B 0,C 180,E1 9786.714,E2 9786.714} C_VEL
LIN {X 0,Y 422.108,Z 688.222,A -85,B 0,C 180,E1 9790.08,E2 9790.08} C_VEL
LIN {X 0,Y 418.409,Z 708.566,A -85,B 0,C 180,E1 9794.307,E2 9794.307} C_VEL
LIN {X 0,Y 415.865,Z 723.504,A -85,B 0,C 180,E1 9798.983,E2 9798.983} C_VEL
LIN {X 0,Y 414.615,Z 732.472,A -85,B 0,C 180,E1 9803.713,E2 9803.713} C_VEL
LIN {X 0,Y 414.051,Z 736.18,A -85,B 0,C 180,E1 9807.906,E2 9807.906} C_VEL
LIN {X 0,Y 414.166,Z 736.119,A -85,B 0,C 180,E1 9812.097,E2 9812.097} C_VEL
LIN {X 0,Y 414.597,Z 732.343,A -85,B 0,C 180,E1 9816.292,E2 9816.292} C_VEL
LIN {X 0,Y 415.899,Z 723.243,A -85,B 0,C 180,E1 9821.02,E2 9821.02} C_VEL
LIN {X 0,Y 418.479,Z 708.098,A -85,B 0,C 180,E1 9825.719,E2 9825.719} C_VEL
LIN {X 0,Y 421.93,Z 689.167,A -85,B 0,C 180,E1 9829.66,E2 9829.66} C_VEL
LIN {X 0,Y 425.939,Z 665.53,A -85,B 0,C 180,E1 9833.157,E2 9833.157} C_VEL
LIN {X 0,Y 430.025,Z 637.538,A -85,B 0,C 180,E1 9836.055,E2 9836.055} C_VEL
LIN {X 0,Y 422.57,Z 610.38,A -85,B 0,C 180,E1 9838.961,E2 9838.961} C_VEL
LIN {X 0,Y 411.288,Z 580.66,A -85,B 0,C 180,E1 9841.787,E2 9841.787} C_VEL
LIN {X 0,Y 411.097,Z 580.66,A -85,B 0,C 180,E1 9848.765,E2 9848.765} C_VEL
LIN {X 0,Y 411.071,Z 580.66,A -85,B 0,C 180,E1 9855.581,E2 9855.581} C_VEL
LIN {X 0,Y 411.062,Z 580.66,A -85,B 0,C 180,E1 9861.226,E2 9861.226} C_VEL
LIN {X 0,Y 411.153,Z 580.66,A -85,B 0,C 180,E1 9867.885,E2 9867.885} C_VEL
LIN {X 0,Y 411.36,Z 580.66,A -85,B 0,C 180,E1 9873.783,E2 9873.783} C_VEL
LIN {X 0,Y 411.665,Z 580.66,A -85,B 0,C 180,E1 9880.664,E2 9880.664} C_VEL
LIN {X 0,Y 411.7,Z 580.66,A -85,B 0,C 180,E1 9887.247,E2 9887.247} C_VEL
LIN {X 0,Y 412.147,Z 580.66,A -85,B 0,C 180,E1 9893.667,E2 9893.667} C_VEL
LIN {X 0,Y 412.427,Z 580.66,A -85,B 0,C 180,E1 9899.994,E2 9899.994} C_VEL
LIN {X 0,Y 412.09,Z 580.66,A -85,B 0,C 180,E1 9906.322,E2 9906.322} C_VEL
LIN {X 0,Y 411.838,Z 580.66,A -85,B 0,C 180,E1 9912.737,E2 9912.737} C_VEL
LIN {X 0,Y 411.642,Z 580.66,A -85,B 0,C 180,E1 9919.325,E2 9919.325} C_VEL
LIN {X 0,Y 411.363,Z 580.66,A -85,B 0,C 180,E1 9926.203,E2 9926.203} C_VEL
LIN {X 0,Y 411.194,Z 580.66,A -85,B 0,C 180,E1 9933.518,E2 9933.518} C_VEL
LIN {X 0,Y 411.046,Z 580.66,A -85,B 0,C 180,E1 9939.328,E2 9939.328} C_VEL
LIN {X 0,Y 411.088,Z 580.66,A -85,B 0,C 180,E1 9945.589,E2 9945.589} C_VEL
LIN {X 0,Y 411.163,Z 580.66,A -85,B 0,C 180,E1 9951.814,E2 9951.814} C_VEL
LIN {X 0,Y 431.332,Z 627.729,A -85,B 0,C 180,E1 9954.657,E2 9954.657} C_VEL
LIN {X 0,Y 434.665,Z 637.409,A -85,B 0,C 180,E1 9955.154,E2 9955.154} C_VEL
LIN {X 0,Y 431.824,Z 677.034,A -85,B 0,C 180,E1 9956.404,E2 9956.404} C_VEL
LIN {X 0,Y 428.002,Z 713.654,A -85,B 0,C 180,E1 9958.398,E2 9958.398} C_VEL
LIN {X 0,Y 423.781,Z 748.871,A -85,B 0,C 180,E1 9961.228,E2 9961.228} C_VEL
LIN {X 0,Y 419.756,Z 780.456,A -85,B 0,C 180,E1 9964.78,E2 9964.78} C_VEL
LIN {X 0,Y 416.563,Z 807.98,A -85,B 0,C 180,E1 9968.965,E2 9968.965} C_VEL
LIN {X 0,Y 415.466,Z 817.95,A -85,B 0,C 180,E1 9970.864,E2 9970.864} C_VEL
LIN {X 0,Y 413.846,Z 822.758,A -85,B 0,C 180,E1 9971.858,E2 9971.858} C_VEL
LIN {X 0,Y 406.387,Z 834.183,A -85,B 0,C 180,E1 9974.664,E2 9974.664} C_VEL
LIN {X 0,Y 406.209,Z 835.14,A -85,B 0,C 180,E1 9974.941,E2 9974.941} C_VEL
LIN {X 0,Y 405.456,Z 849.274,A -85,B 0,C 180,E1 9979.781,E2 9979.781} C_VEL
LIN {X 0,Y 405.368,Z 857.85,A -85,B 0,C 180,E1 9984.64,E2 9984.64} C_VEL
LIN {X 0,Y 405.303,Z 860.556,A -85,B 0,C 180,E1 9987.857,E2 9987.857} C_VEL
LIN {X 0,Y 405.331,Z 860.563,A -85,B 0,C 180,E1 9992.139,E2 9992.139} C_VEL
LIN {X 0,Y 405.352,Z 856.476,A -85,B 0,C 180,E1 9996.432,E2 9996.432} C_VEL
LIN {X 0,Y 405.596,Z 846.659,A -85,B 0,C 180,E1 10001.3,E2 10001.3} C_VEL
LIN {X 0,Y 406.539,Z 830.87,A -85,B 0,C 180,E1 10006.217,E2 10006.217} C_VEL
LIN {X 0,Y 408.598,Z 809.56,A -85,B 0,C 180,E1 10010.892,E2 10010.892} C_VEL
LIN {X 0,Y 411.953,Z 782.126,A -85,B 0,C 180,E1 10015.291,E2 10015.291} C_VEL
LIN {X 0,Y 415.941,Z 752.441,A -85,B 0,C 180,E1 10018.8,E2 10018.8} C_VEL
LIN {X 0,Y 420.324,Z 718.047,A -85,B 0,C 180,E1 10021.771,E2 10021.771} C_VEL
LIN {X 0,Y 424.592,Z 680.868,A -85,B 0,C 180,E1 10023.934,E2 10023.934} C_VEL
LIN {X 0,Y 427.779,Z 642.857,A -85,B 0,C 180,E1 10025.262,E2 10025.262} C_VEL
LIN {X 0,Y 425.788,Z 633.259,A -85,B 0,C 180,E1 10025.682,E2 10025.682} C_VEL
LIN {X 0,Y 411.515,Z 599.014,A -85,B 0,C 180,E1 10027.729,E2 10027.729} C_VEL
LIN {X 0,Y 403.153,Z 580.66,A -85,B 0,C 180,E1 10029.009,E2 10029.009} C_VEL
LIN {X 0,Y 403.189,Z 580.66,A -85,B 0,C 180,E1 10035.515,E2 10035.515} C_VEL
LIN {X 0,Y 403.133,Z 580.66,A -85,B 0,C 180,E1 10042.059,E2 10042.059} C_VEL
LIN {X 0,Y 403.283,Z 580.66,A -85,B 0,C 180,E1 10048.299,E2 10048.299} C_VEL
LIN {X 0,Y 403.467,Z 580.66,A -85,B 0,C 180,E1 10055.627,E2 10055.627} C_VEL
LIN {X 0,Y 403.729,Z 580.66,A -85,B 0,C 180,E1 10062.548,E2 10062.548} C_VEL
LIN {X 0,Y 403.876,Z 580.66,A -85,B 0,C 180,E1 10069.203,E2 10069.203} C_VEL
LIN {X 0,Y 404.232,Z 580.66,A -85,B 0,C 180,E1 10075.71,E2 10075.71} C_VEL
LIN {X 0,Y 404.461,Z 580.66,A -85,B 0,C 180,E1 10082.151,E2 10082.151} C_VEL
LIN {X 0,Y 404.095,Z 580.66,A -85,B 0,C 180,E1 10088.625,E2 10088.625} C_VEL
LIN {X 0,Y 403.826,Z 580.66,A -85,B 0,C 180,E1 10095.221,E2 10095.221} C_VEL
LIN {X 0,Y 403.581,Z 580.66,A -85,B 0,C 180,E1 10102.04,E2 10102.04} C_VEL
LIN {X 0,Y 403.355,Z 580.66,A -85,B 0,C 180,E1 10109.214,E2 10109.214} C_VEL
LIN {X 0,Y 403.27,Z 580.66,A -85,B 0,C 180,E1 10114.318,E2 10114.318} C_VEL
LIN {X 0,Y 403.086,Z 580.66,A -85,B 0,C 180,E1 10121.307,E2 10121.307} C_VEL
LIN {X 0,Y 403.092,Z 580.66,A -85,B 0,C 180,E1 10128.704,E2 10128.704} C_VEL
LIN {X 0,Y 403.315,Z 580.66,A -85,B 0,C 180,E1 10135.733,E2 10135.733} C_VEL
LIN {X 0,Y 403.408,Z 580.66,A -85,B 0,C 180,E1 10137.409,E2 10137.409} C_VEL
LIN {X 0,Y 415.408,Z 612.196,A -85,B 0,C 180,E1 10140.395,E2 10140.395} C_VEL
LIN {X 0,Y 422.97,Z 639.804,A -85,B 0,C 180,E1 10143.455,E2 10143.455} C_VEL
LIN {X 0,Y 418.726,Z 667.58,A -85,B 0,C 180,E1 10146.424,E2 10146.424} C_VEL
LIN {X 0,Y 414.503,Z 690.995,A -85,B 0,C 180,E1 10149.977,E2 10149.977} C_VEL
LIN {X 0,Y 410.871,Z 709.843,A -85,B 0,C 180,E1 10154.024,E2 10154.024} C_VEL
LIN {X 0,Y 408.198,Z 724.712,A -85,B 0,C 180,E1 10158.773,E2 10158.773} C_VEL
LIN {X 0,Y 406.836,Z 733.666,A -85,B 0,C 180,E1 10163.592,E2 10163.592} C_VEL
LIN {X 0,Y 406.251,Z 737.367,A -85,B 0,C 180,E1 10167.866,E2 10167.866} C_VEL
LIN {X 0,Y 406.357,Z 737.307,A -85,B 0,C 180,E1 10172.137,E2 10172.137} C_VEL
LIN {X 0,Y 406.82,Z 733.538,A -85,B 0,C 180,E1 10176.412,E2 10176.412} C_VEL
LIN {X 0,Y 408.25,Z 724.452,A -85,B 0,C 180,E1 10181.229,E2 10181.229} C_VEL
LIN {X 0,Y 410.95,Z 709.366,A -85,B 0,C 180,E1 10186.006,E2 10186.006} C_VEL
LIN {X 0,Y 414.594,Z 690.443,A -85,B 0,C 180,E1 10190.023,E2 10190.023} C_VEL
LIN {X 0,Y 418.797,Z 666.859,A -85,B 0,C 180,E1 10193.576,E2 10193.576} C_VEL
LIN {X 0,Y 423.063,Z 638.972,A -85,B 0,C 180,E1 10196.519,E2 10196.519} C_VEL
LIN {X 0,Y 414.641,Z 609.793,A -85,B 0,C 180,E1 10199.75,E2 10199.75} C_VEL
LIN {X 0,Y 403.331,Z 580.66,A -85,B 0,C 180,E1 10202.525,E2 10202.525} C_VEL
LIN {X 0,Y 403.15,Z 580.66,A -85,B 0,C 180,E1 10209.677,E2 10209.677} C_VEL
LIN {X 0,Y 403.167,Z 580.66,A -85,B 0,C 180,E1 10215.524,E2 10215.524} C_VEL
LIN {X 0,Y 403.084,Z 580.66,A -85,B 0,C 180,E1 10222.075,E2 10222.075} C_VEL
LIN {X 0,Y 403.263,Z 580.66,A -85,B 0,C 180,E1 10228.283,E2 10228.283} C_VEL
LIN {X 0,Y 403.486,Z 580.66,A -85,B 0,C 180,E1 10235.615,E2 10235.615} C_VEL
LIN {X 0,Y 403.73,Z 580.66,A -85,B 0,C 180,E1 10242.536,E2 10242.536} C_VEL
LIN {X 0,Y 403.854,Z 580.66,A -85,B 0,C 180,E1 10249.19,E2 10249.19} C_VEL
LIN {X 0,Y 404.263,Z 580.66,A -85,B 0,C 180,E1 10255.698,E2 10255.698} C_VEL
LIN {X 0,Y 404.41,Z 580.66,A -85,B 0,C 180,E1 10262.14,E2 10262.14} C_VEL
LIN {X 0,Y 404.107,Z 580.66,A -85,B 0,C 180,E1 10268.613,E2 10268.613} C_VEL
LIN {X 0,Y 403.83,Z 580.66,A -85,B 0,C 180,E1 10275.209,E2 10275.209} C_VEL
LIN {X 0,Y 403.603,Z 580.66,A -85,B 0,C 180,E1 10282.026,E2 10282.026} C_VEL
LIN {X 0,Y 403.326,Z 580.66,A -85,B 0,C 180,E1 10289.202,E2 10289.202} C_VEL
LIN {X 0,Y 403.226,Z 580.66,A -85,B 0,C 180,E1 10294.302,E2 10294.302} C_VEL
LIN {X 0,Y 403.113,Z 580.66,A -85,B 0,C 180,E1 10301.306,E2 10301.306} C_VEL
LIN {X 0,Y 403.186,Z 580.66,A -85,B 0,C 180,E1 10307.471,E2 10307.471} C_VEL
LIN {X 0,Y 403.227,Z 581.064,A -85,B 0,C 180,E1 10311.055,E2 10311.055} C_VEL
LIN {X 0,Y 423.829,Z 627.669,A -85,B 0,C 180,E1 10314.022,E2 10314.022} C_VEL
LIN {X 0,Y 427.862,Z 640.994,A -85,B 0,C 180,E1 10314.692,E2 10314.692} C_VEL
LIN {X 0,Y 424.709,Z 679.27,A -85,B 0,C 180,E1 10315.995,E2 10315.995} C_VEL
LIN {X 0,Y 420.521,Z 716.596,A -85,B 0,C 180,E1 10318.131,E2 10318.131} C_VEL
LIN {X 0,Y 416.099,Z 750.874,A -85,B 0,C 180,E1 10321.042,E2 10321.042} C_VEL
LIN {X 0,Y 411.949,Z 782.078,A -85,B 0,C 180,E1 10324.705,E2 10324.705} C_VEL
LIN {X 0,Y 408.623,Z 809.539,A -85,B 0,C 180,E1 10329.105,E2 10329.105} C_VEL
LIN {X 0,Y 406.537,Z 830.853,A -85,B 0,C 180,E1 10333.779,E2 10333.779} C_VEL
LIN {X 0,Y 406.209,Z 835.14,A -85,B 0,C 180,E1 10334.941,E2 10334.941} C_VEL
LIN {X 0,Y 404.665,Z 838.844,A -85,B 0,C 180,E1 10336.046,E2 10336.046} C_VEL
LIN {X 0,Y 397.731,Z 847.064,A -85,B 0,C 180,E1 10339.158,E2 10339.158} C_VEL
LIN {X 0,Y 397.631,Z 847.747,A -85,B 0,C 180,E1 10339.458,E2 10339.458} C_VEL
LIN {X 0,Y 397.544,Z 855.257,A -85,B 0,C 180,E1 10343.437,E2 10343.437} C_VEL
LIN {X 0,Y 397.482,Z 859.365,A -85,B 0,C 180,E1 10347.815,E2 10347.815} C_VEL
LIN {X 0,Y 397.509,Z 859.372,A -85,B 0,C 180,E1 10352.181,E2 10352.181} C_VEL
LIN {X 0,Y 397.535,Z 855.264,A -85,B 0,C 180,E1 10356.559,E2 10356.559} C_VEL
LIN {X 0,Y 397.746,Z 845.394,A -85,B 0,C 180,E1 10361.526,E2 10361.526} C_VEL
LIN {X 0,Y 398.774,Z 829.56,A -85,B 0,C 180,E1 10366.542,E2 10366.542} C_VEL
LIN {X 0,Y 400.877,Z 808.184,A -85,B 0,C 180,E1 10371.314,E2 10371.314} C_VEL
LIN {X 0,Y 404.446,Z 781.135,A -85,B 0,C 180,E1 10375.729,E2 10375.729} C_VEL
LIN {X 0,Y 408.802,Z 750.669,A -85,B 0,C 180,E1 10379.381,E2 10379.381} C_VEL
LIN {X 0,Y 413.516,Z 716.023,A -85,B 0,C 180,E1 10382.391,E2 10382.391} C_VEL
LIN {X 0,Y 417.815,Z 679.439,A -85,B 0,C 180,E1 10384.531,E2 10384.531} C_VEL
LIN {X 0,Y 420.949,Z 641.153,A -85,B 0,C 180,E1 10385.887,E2 10385.887} C_VEL
LIN {X 0,Y 407.71,Z 607.378,A -85,B 0,C 180,E1 10387.907,E2 10387.907} C_VEL
LIN {X 0,Y 395.208,Z 580.66,A -85,B 0,C 180,E1 10389.917,E2 10389.917} C_VEL
LIN {X 0,Y 395.258,Z 580.66,A -85,B 0,C 180,E1 10396.698,E2 10396.698} C_VEL
LIN {X 0,Y 395.218,Z 580.66,A -85,B 0,C 180,E1 10403.556,E2 10403.556} C_VEL
LIN {X 0,Y 395.398,Z 580.66,A -85,B 0,C 180,E1 10410.153,E2 10410.153} C_VEL
LIN {X 0,Y 395.62,Z 580.66,A -85,B 0,C 180,E1 10417.506,E2 10417.506} C_VEL
LIN {X 0,Y 395.792,Z 580.66,A -85,B 0,C 180,E1 10424.475,E2 10424.475} C_VEL
LIN {X 0,Y 396.136,Z 580.66,A -85,B 0,C 180,E1 10431.212,E2 10431.212} C_VEL
LIN {X 0,Y 396.59,Z 580.66,A -85,B 0,C 180,E1 10437.818,E2 10437.818} C_VEL
LIN {X 0,Y 396.424,Z 580.66,A -85,B 0,C 180,E1 10444.387,E2 10444.387} C_VEL
LIN {X 0,Y 396.032,Z 580.66,A -85,B 0,C 180,E1 10451.026,E2 10451.026} C_VEL
LIN {X 0,Y 395.848,Z 580.66,A -85,B 0,C 180,E1 10457.824,E2 10457.824} C_VEL
LIN {X 0,Y 395.533,Z 580.66,A -85,B 0,C 180,E1 10464.908,E2 10464.908} C_VEL
LIN {X 0,Y 395.431,Z 580.66,A -85,B 0,C 180,E1 10469.858,E2 10469.858} C_VEL
LIN {X 0,Y 395.251,Z 580.66,A -85,B 0,C 180,E1 10476.45,E2 10476.45} C_VEL
LIN {X 0,Y 395.125,Z 580.66,A -85,B 0,C 180,E1 10483.281,E2 10483.281} C_VEL
LIN {X 0,Y 395.225,Z 580.66,A -85,B 0,C 180,E1 10490.02,E2 10490.02} C_VEL
LIN {X 0,Y 395.482,Z 581.24,A -85,B 0,C 180,E1 10496.587,E2 10496.587} C_VEL
LIN {X 0,Y 407.86,Z 612.518,A -85,B 0,C 180,E1 10499.679,E2 10499.679} C_VEL
LIN {X 0,Y 415.723,Z 640.435,A -85,B 0,C 180,E1 10502.866,E2 10502.866} C_VEL
LIN {X 0,Y 411.623,Z 668.893,A -85,B 0,C 180,E1 10505.992,E2 10505.992} C_VEL
LIN {X 0,Y 407.168,Z 692.265,A -85,B 0,C 180,E1 10509.6,E2 10509.6} C_VEL
LIN {X 0,Y 403.238,Z 711.698,A -85,B 0,C 180,E1 10513.889,E2 10513.889} C_VEL
LIN {X 0,Y 400.541,Z 725.917,A -85,B 0,C 180,E1 10518.556,E2 10518.556} C_VEL
LIN {X 0,Y 399.09,Z 734.855,A -85,B 0,C 180,E1 10523.467,E2 10523.467} C_VEL
LIN {X 0,Y 398.468,Z 738.55,A -85,B 0,C 180,E1 10527.824,E2 10527.824} C_VEL
LIN {X 0,Y 398.572,Z 738.491,A -85,B 0,C 180,E1 10532.179,E2 10532.179} C_VEL
LIN {X 0,Y 399.074,Z 734.729,A -85,B 0,C 180,E1 10536.537,E2 10536.537} C_VEL
LIN {X 0,Y 400.587,Z 725.662,A -85,B 0,C 180,E1 10541.447,E2 10541.447} C_VEL
LIN {X 0,Y 403.314,Z 711.233,A -85,B 0,C 180,E1 10546.139,E2 10546.139} C_VEL
LIN {X 0,Y 407.276,Z 691.716,A -85,B 0,C 180,E1 10550.398,E2 10550.398} C_VEL
LIN {X 0,Y 411.933,Z 667.165,A -85,B 0,C 180,E1 10554.137,E2 10554.137} C_VEL
LIN {X 0,Y 415.768,Z 640.5,A -85,B 0,C 180,E1 10557.022,E2 10557.022} C_VEL
LIN {X 0,Y 407.829,Z 612.584,A -85,B 0,C 180,E1 10560.216,E2 10560.216} C_VEL
LIN {X 0,Y 396.032,Z 583.751,A -85,B 0,C 180,E1 10563.142,E2 10563.142} C_VEL
LIN {X 0,Y 395.357,Z 580.66,A -85,B 0,C 180,E1 10563.474,E2 10563.474} C_VEL
LIN {X 0,Y 395.229,Z 580.66,A -85,B 0,C 180,E1 10570.637,E2 10570.637} C_VEL
LIN {X 0,Y 395.209,Z 580.66,A -85,B 0,C 180,E1 10576.712,E2 10576.712} C_VEL
LIN {X 0,Y 395.165,Z 580.66,A -85,B 0,C 180,E1 10583.574,E2 10583.574} C_VEL
LIN {X 0,Y 395.394,Z 580.66,A -85,B 0,C 180,E1 10590.139,E2 10590.139} C_VEL
LIN {X 0,Y 395.637,Z 580.66,A -85,B 0,C 180,E1 10597.494,E2 10597.494} C_VEL
LIN {X 0,Y 395.779,Z 580.66,A -85,B 0,C 180,E1 10604.461,E2 10604.461} C_VEL
LIN {X 0,Y 396.139,Z 580.66,A -85,B 0,C 180,E1 10611.556,E2 10611.556} C_VEL
LIN {X 0,Y 396.621,Z 580.66,A -85,B 0,C 180,E1 10617.806,E2 10617.806} C_VEL
LIN {X 0,Y 396.422,Z 580.66,A -85,B 0,C 180,E1 10624.375,E2 10624.375} C_VEL
LIN {X 0,Y 396.046,Z 580.66,A -85,B 0,C 180,E1 10631.013,E2 10631.013} C_VEL
LIN {X 0,Y 395.85,Z 580.66,A -85,B 0,C 180,E1 10637.811,E2 10637.811} C_VEL
LIN {X 0,Y 395.533,Z 580.66,A -85,B 0,C 180,E1 10644.895,E2 10644.895} C_VEL
LIN {X 0,Y 395.398,Z 580.66,A -85,B 0,C 180,E1 10649.847,E2 10649.847} C_VEL
LIN {X 0,Y 395.182,Z 580.66,A -85,B 0,C 180,E1 10656.43,E2 10656.43} C_VEL
LIN {X 0,Y 395.218,Z 580.66,A -85,B 0,C 180,E1 10663.587,E2 10663.587} C_VEL
LIN {X 0,Y 395.255,Z 580.66,A -85,B 0,C 180,E1 10670.208,E2 10670.208} C_VEL
LIN {X 0,Y 417.056,Z 629.599,A -85,B 0,C 180,E1 10673.474,E2 10673.474} C_VEL
LIN {X 0,Y 420.987,Z 643.492,A -85,B 0,C 180,E1 10674.198,E2 10674.198} C_VEL
LIN {X 0,Y 417.524,Z 682.126,A -85,B 0,C 180,E1 10675.597,E2 10675.597} C_VEL
LIN {X 0,Y 413.045,Z 719.236,A -85,B 0,C 180,E1 10677.854,E2 10677.854} C_VEL
